   AI_RAW_7801.___________0020_1 := false;
   AI_RAW_7801.RAW_MIN := -6000;
   AI_RAW_7801.RAW_MAX := 13000;
   AI_RAW_7801.RAW_DESC := 'Thermal Resistance - 4-wire (Ni100 climate - 618)';
   AI_RAW_7801.___________0030_1 := false;
   AI_RAW_7801.___________0030_2 := false;
   AI_RAW_7801.PARAM_TYPE := 16#07;
   AI_RAW_7801.PARAM_RANGE := 16#01;
   AI_RAW_7801.PARAM_COEF := 16#08;
   AI_RAW_7801.___________0040_1 := false;
   AI_RAW_7801.___________0040_2 := false;
   AI_RAW_7801.VALUE_COEF := 0.00618;
   AI_RAW_7901.revInfo.REV_BLOCK := 'UT00801';
   AI_RAW_7901.revInfo.REV_NUMBER := '001.000';
   AI_RAW_7901.revInfo.REV_DATE := '2024-04-09';
   AI_RAW_7901.revInfo.REV_AUTHOR := 'M. Gledhill';
   AI_RAW_7901.___________0010_0 := false;
   AI_RAW_7901.___________0010_1 := false;
   AI_RAW_7901.AI_CODE := 16#7901;
   AI_RAW_7901.___________0020_0 := false;
   AI_RAW_7901.___________0020_1 := false;
   AI_RAW_7901.RAW_MIN := -6000;
   AI_RAW_7901.RAW_MAX := 13000;
   AI_RAW_7901.RAW_DESC := 'Thermal Resistance - 4-wire (Ni100 climate - 672)';
   AI_RAW_7901.___________0030_1 := false;
   AI_RAW_7901.___________0030_2 := false;
   AI_RAW_7901.PARAM_TYPE := 16#07;
   AI_RAW_7901.PARAM_RANGE := 16#01;
   AI_RAW_7901.PARAM_COEF := 16#09;
   AI_RAW_7901.___________0040_1 := false;
   AI_RAW_7901.___________0040_2 := false;
   AI_RAW_7901.VALUE_COEF := 0.00672;
   AI_RAW_7703.revInfo.REV_BLOCK := 'UT00801';
   AI_RAW_7703.revInfo.REV_NUMBER := '001.000';
   AI_RAW_7703.revInfo.REV_DATE := '2024-04-09';
   AI_RAW_7703.revInfo.REV_AUTHOR := 'M. Gledhill';
   AI_RAW_7703.___________0010_0 := false;
   AI_RAW_7703.___________0010_1 := false;
   AI_RAW_7703.AI_CODE := 16#7703;
   AI_RAW_7703.___________0020_0 := false;
   AI_RAW_7703.___________0020_1 := false;
   AI_RAW_7703.RAW_MIN := -600;
   AI_RAW_7703.RAW_MAX := 1800;
   AI_RAW_7703.RAW_DESC := 'Thermal Resistance - 4-wire (Ni100 standard - 617)';
   AI_RAW_7703.___________0030_1 := false;
   AI_RAW_7703.___________0030_2 := false;
   AI_RAW_7703.PARAM_TYPE := 16#07;
   AI_RAW_7703.PARAM_RANGE := 16#03;
   AI_RAW_7703.PARAM_COEF := 16#07;
   AI_RAW_7703.___________0040_1 := false;
   AI_RAW_7703.___________0040_2 := false;
   AI_RAW_7703.VALUE_COEF := 0.00617;
   AI_RAW_7803.revInfo.REV_BLOCK := 'UT00801';
   AI_RAW_7803.revInfo.REV_NUMBER := '001.000';
   AI_RAW_7803.revInfo.REV_DATE := '2024-04-09';
   AI_RAW_7803.revInfo.REV_AUTHOR := 'M. Gledhill';
   AI_RAW_7803.___________0010_0 := false;
   AI_RAW_7803.___________0010_1 := false;
   AI_RAW_7803.AI_CODE := 16#7803;
   AI_RAW_7803.___________0020_0 := false;
   AI_RAW_7803.___________0020_1 := false;
   AI_RAW_7803.RAW_MIN := -600;
   AI_RAW_7803.RAW_MAX := 2500;
   AI_RAW_7803.RAW_DESC := 'Thermal Resistance - 4-wire (Ni100 standard - 618)';
   AI_RAW_7803.___________0030_1 := false;
   AI_RAW_7803.___________0030_2 := false;
   AI_RAW_7803.PARAM_TYPE := 16#07;
   AI_RAW_7803.PARAM_RANGE := 16#03;
   AI_RAW_7803.PARAM_COEF := 16#08;
   AI_RAW_7803.___________0040_1 := false;
   AI_RAW_7803.___________0040_2 := false;
   AI_RAW_7803.VALUE_COEF := 0.00618;
   AI_RAW_7903.revInfo.REV_BLOCK := 'UT00801';
   AI_RAW_7903.revInfo.REV_NUMBER := '001.000';
   AI_RAW_7903.revInfo.REV_DATE := '2024-04-09';
   AI_RAW_7903.revInfo.REV_AUTHOR := 'M. Gledhill';
   AI_RAW_7903.___________0010_0 := false;
   AI_RAW_7903.___________0010_1 := false;
   AI_RAW_7903.AI_CODE := 16#7903;
   AI_RAW_7903.___________0020_0 := false;
   AI_RAW_7903.___________0020_1 := false;
   AI_RAW_7903.RAW_MIN := -600;
   AI_RAW_7903.RAW_MAX := 2500;
   AI_RAW_7903.RAW_DESC := 'Thermal Resistance - 4-wire (Ni100 standard - 672)';
   AI_RAW_7903.___________0030_1 := false;
   AI_RAW_7903.___________0030_2 := false;
   AI_RAW_7903.PARAM_TYPE := 16#07;
   AI_RAW_7903.PARAM_RANGE := 16#03;
   AI_RAW_7903.PARAM_COEF := 16#09;
   AI_RAW_7903.___________0040_1 := false;
   AI_RAW_7903.___________0040_2 := false;
   AI_RAW_7903.VALUE_COEF := 0.00672;
   AI_RAW_7711.revInfo.REV_BLOCK := 'UT00801';
   AI_RAW_7711.revInfo.REV_NUMBER := '001.000';
   AI_RAW_7711.revInfo.REV_DATE := '2024-04-09';
   AI_RAW_7711.revInfo.REV_AUTHOR := 'M. Gledhill';
   AI_RAW_7711.___________0010_0 := false;
   AI_RAW_7711.___________0010_1 := false;
   AI_RAW_7711.AI_CODE := 16#7711;
   AI_RAW_7711.___________0020_0 := false;
   AI_RAW_7711.___________0020_1 := false;
   AI_RAW_7711.RAW_MIN := -6000;
   AI_RAW_7711.RAW_MAX := 13000;
   AI_RAW_7711.RAW_DESC := 'Thermal Resistance - 4-wire (Ni200 climate - 617)';
   AI_RAW_7711.___________0030_1 := false;
   AI_RAW_7711.___________0030_2 := false;
   AI_RAW_7711.PARAM_TYPE := 16#07;
   AI_RAW_7711.PARAM_RANGE := 16#11;
   AI_RAW_7711.PARAM_COEF := 16#07;
   AI_RAW_7711.___________0040_1 := false;
   AI_RAW_7711.___________0040_2 := false;
   AI_RAW_7711.VALUE_COEF := 0.00617;
   AI_RAW_7811.revInfo.REV_BLOCK := 'UT00801';
   AI_RAW_7811.revInfo.REV_NUMBER := '001.000';
   AI_RAW_7811.revInfo.REV_DATE := '2024-04-09';
   AI_RAW_7811.revInfo.REV_AUTHOR := 'M. Gledhill';
   AI_RAW_7811.___________0010_0 := false;
   AI_RAW_7811.___________0010_1 := false;
   AI_RAW_7811.AI_CODE := 16#7811;
   AI_RAW_7811.___________0020_0 := false;
   AI_RAW_7811.___________0020_1 := false;
   AI_RAW_7811.RAW_MIN := -6000;
   AI_RAW_7811.RAW_MAX := 13000;
   AI_RAW_7811.RAW_DESC := 'Thermal Resistance - 4-wire (Ni200 climate - 618)';
   AI_RAW_7811.___________0030_1 := false;
   AI_RAW_7811.___________0030_2 := false;
   AI_RAW_7811.PARAM_TYPE := 16#07;
   AI_RAW_7811.PARAM_RANGE := 16#11;
   AI_RAW_7811.PARAM_COEF := 16#08;
   AI_RAW_7811.___________0040_1 := false;
   AI_RAW_7811.___________0040_2 := false;
   AI_RAW_7811.VALUE_COEF := 0.00618;
   AI_RAW_7911.revInfo.REV_BLOCK := 'UT00801';
   AI_RAW_7911.revInfo.REV_NUMBER := '001.000';
   AI_RAW_7911.revInfo.REV_DATE := '2024-04-09';
   AI_RAW_7911.revInfo.REV_AUTHOR := 'M. Gledhill';
   AI_RAW_7911.___________0010_0 := false;
   AI_RAW_7911.___________0010_1 := false;
   AI_RAW_7911.AI_CODE := 16#7911;
   AI_RAW_7911.___________0020_0 := false;
   AI_RAW_7911.___________0020_1 := false;
   AI_RAW_7911.RAW_MIN := -6000;
   AI_RAW_7911.RAW_MAX := 13000;
   AI_RAW_7911.RAW_DESC := 'Thermal Resistance - 4-wire (Ni200 climate - 672)';
   AI_RAW_7911.___________0030_1 := false;
   AI_RAW_7911.___________0030_2 := false;
   AI_RAW_7911.PARAM_TYPE := 16#07;
   AI_RAW_7911.PARAM_RANGE := 16#11;
   AI_RAW_7911.PARAM_COEF := 16#09;
   AI_RAW_7911.___________0040_1 := false;
   AI_RAW_7911.___________0040_2 := false;
   AI_RAW_7911.VALUE_COEF := 0.00672;
   AI_RAW_7710.revInfo.REV_BLOCK := 'UT00801';
   AI_RAW_7710.revInfo.REV_NUMBER := '001.000';
   AI_RAW_7710.revInfo.REV_DATE := '2024-04-09';
   AI_RAW_7710.revInfo.REV_AUTHOR := 'M. Gledhill';
   AI_RAW_7710.___________0010_0 := false;
   AI_RAW_7710.___________0010_1 := false;
   AI_RAW_7710.AI_CODE := 16#7710;
   AI_RAW_7710.___________0020_0 := false;
   AI_RAW_7710.___________0020_1 := false;
   AI_RAW_7710.RAW_MIN := -600;
   AI_RAW_7710.RAW_MAX := 1800;
   AI_RAW_7710.RAW_DESC := 'Thermal Resistance - 4-wire (Ni200 standard - 617)';
   AI_RAW_7710.___________0030_1 := false;
   AI_RAW_7710.___________0030_2 := false;
   AI_RAW_7710.PARAM_TYPE := 16#07;
   AI_RAW_7710.PARAM_RANGE := 16#10;
   AI_RAW_7710.PARAM_COEF := 16#07;
   AI_RAW_7710.___________0040_1 := false;
   AI_RAW_7710.___________0040_2 := false;
   AI_RAW_7710.VALUE_COEF := 0.00617;
   AI_RAW_7810.revInfo.REV_BLOCK := 'UT00801';
   AI_RAW_7810.revInfo.REV_NUMBER := '001.000';
   AI_RAW_7810.revInfo.REV_DATE := '2024-04-09';
   AI_RAW_7810.revInfo.REV_AUTHOR := 'M. Gledhill';
   AI_RAW_7810.___________0010_0 := false;
   AI_RAW_7810.___________0010_1 := false;
   AI_RAW_7810.AI_CODE := 16#7810;
   AI_RAW_7810.___________0020_0 := false;
   AI_RAW_7810.___________0020_1 := false;
   AI_RAW_7810.RAW_MIN := -600;
   AI_RAW_7810.RAW_MAX := 2500;
   AI_RAW_7810.RAW_DESC := 'Thermal Resistance - 4-wire (Ni200 standard - 618)';
   AI_RAW_7810.___________0030_1 := false;
   AI_RAW_7810.___________0030_2 := false;
   AI_RAW_7810.PARAM_TYPE := 16#07;
   AI_RAW_7810.PARAM_RANGE := 16#10;
   AI_RAW_7810.PARAM_COEF := 16#08;
   AI_RAW_7810.___________0040_1 := false;
   AI_RAW_7810.___________0040_2 := false;
   AI_RAW_7810.VALUE_COEF := 0.00618;
   AI_RAW_7910.revInfo.REV_BLOCK := 'UT00801';
   AI_RAW_7910.revInfo.REV_NUMBER := '001.000';
   AI_RAW_7910.revInfo.REV_DATE := '2024-04-09';
   AI_RAW_7910.revInfo.REV_AUTHOR := 'M. Gledhill';
   AI_RAW_7910.___________0010_0 := false;
   AI_RAW_7910.___________0010_1 := false;
   AI_RAW_7910.AI_CODE := 16#7910;
   AI_RAW_7910.___________0020_0 := false;
   AI_RAW_7910.___________0020_1 := false;
   AI_RAW_7910.RAW_MIN := -600;
   AI_RAW_7910.RAW_MAX := 2500;
   AI_RAW_7910.RAW_DESC := 'Thermal Resistance - 4-wire (Ni200 standard - 672)';
   AI_RAW_7910.___________0030_1 := false;
   AI_RAW_7910.___________0030_2 := false;
   AI_RAW_7910.PARAM_TYPE := 16#07;
   AI_RAW_7910.PARAM_RANGE := 16#10;
   AI_RAW_7910.PARAM_COEF := 16#09;
   AI_RAW_7910.___________0040_1 := false;
   AI_RAW_7910.___________0040_2 := false;
   AI_RAW_7910.VALUE_COEF := 0.00672;
   AI_RAW_7713.revInfo.REV_BLOCK := 'UT00801';
   AI_RAW_7713.revInfo.REV_NUMBER := '001.000';
   AI_RAW_7713.revInfo.REV_DATE := '2024-04-09';
   AI_RAW_7713.revInfo.REV_AUTHOR := 'M. Gledhill';
   AI_RAW_7713.___________0010_0 := false;
   AI_RAW_7713.___________0010_1 := false;
   AI_RAW_7713.AI_CODE := 16#7713;
   AI_RAW_7713.___________0020_0 := false;
   AI_RAW_7713.___________0020_1 := false;
   AI_RAW_7713.RAW_MIN := -6000;
   AI_RAW_7713.RAW_MAX := 13000;
   AI_RAW_7713.RAW_DESC := 'Thermal Resistance - 4-wire (Ni500 climate - 617)';
   AI_RAW_7713.___________0030_1 := false;
   AI_RAW_7713.___________0030_2 := false;
   AI_RAW_7713.PARAM_TYPE := 16#07;
   AI_RAW_7713.PARAM_RANGE := 16#13;
   AI_RAW_7713.PARAM_COEF := 16#07;
   AI_RAW_7713.___________0040_1 := false;
   AI_RAW_7713.___________0040_2 := false;
   AI_RAW_7713.VALUE_COEF := 0.00617;
   AI_RAW_7813.revInfo.REV_BLOCK := 'UT00801';
   AI_RAW_7813.revInfo.REV_NUMBER := '001.000';
   AI_RAW_7813.revInfo.REV_DATE := '2024-04-09';
   AI_RAW_7813.revInfo.REV_AUTHOR := 'M. Gledhill';
   AI_RAW_7813.___________0010_0 := false;
   AI_RAW_7813.___________0010_1 := false;
   AI_RAW_7813.AI_CODE := 16#7813;
   AI_RAW_7813.___________0020_0 := false;
   AI_RAW_7813.___________0020_1 := false;
   AI_RAW_7813.RAW_MIN := -6000;
   AI_RAW_7813.RAW_MAX := 13000;
   AI_RAW_7813.RAW_DESC := 'Thermal Resistance - 4-wire (Ni500 climate - 618)';
   AI_RAW_7813.___________0030_1 := false;
   AI_RAW_7813.___________0030_2 := false;
   AI_RAW_7813.PARAM_TYPE := 16#07;
   AI_RAW_7813.PARAM_RANGE := 16#13;
   AI_RAW_7813.PARAM_COEF := 16#08;
   AI_RAW_7813.___________0040_1 := false;
   AI_RAW_7813.___________0040_2 := false;
   AI_RAW_7813.VALUE_COEF := 0.00618;
   AI_RAW_7913.revInfo.REV_BLOCK := 'UT00801';
   AI_RAW_7913.revInfo.REV_NUMBER := '001.000';
   AI_RAW_7913.revInfo.REV_DATE := '2024-04-09';
   AI_RAW_7913.revInfo.REV_AUTHOR := 'M. Gledhill';
   AI_RAW_7913.___________0010_0 := false;
   AI_RAW_7913.___________0010_1 := false;
   AI_RAW_7913.AI_CODE := 16#7913;
   AI_RAW_7913.___________0020_0 := false;
   AI_RAW_7913.___________0020_1 := false;
   AI_RAW_7913.RAW_MIN := -6000;
   AI_RAW_7913.RAW_MAX := 13000;
   AI_RAW_7913.RAW_DESC := 'Thermal Resistance - 4-wire (Ni500 climate - 672)';
   AI_RAW_7913.___________0030_1 := false;
   AI_RAW_7913.___________0030_2 := false;
   AI_RAW_7913.PARAM_TYPE := 16#07;
   AI_RAW_7913.PARAM_RANGE := 16#13;
   AI_RAW_7913.PARAM_COEF := 16#09;
   AI_RAW_7913.___________0040_1 := false;
   AI_RAW_7913.___________0040_2 := false;
   AI_RAW_7913.VALUE_COEF := 0.00672;
   AI_RAW_7712.revInfo.REV_BLOCK := 'UT00801';
   AI_RAW_7712.revInfo.REV_NUMBER := '001.000';
   AI_RAW_7712.revInfo.REV_DATE := '2024-04-09';
   AI_RAW_7712.revInfo.REV_AUTHOR := 'M. Gledhill';
   AI_RAW_7712.___________0010_0 := false;
   AI_RAW_7712.___________0010_1 := false;
   AI_RAW_7712.AI_CODE := 16#7712;
   AI_RAW_7712.___________0020_0 := false;
   AI_RAW_7712.___________0020_1 := false;
   AI_RAW_7712.RAW_MIN := -600;
   AI_RAW_7712.RAW_MAX := 1800;
   AI_RAW_7712.RAW_DESC := 'Thermal Resistance - 4-wire (Ni500 standard - 617)';
   AI_RAW_7712.___________0030_1 := false;
   AI_RAW_7712.___________0030_2 := false;
   AI_RAW_7712.PARAM_TYPE := 16#07;
   AI_RAW_7712.PARAM_RANGE := 16#12;
   AI_RAW_7712.PARAM_COEF := 16#07;
   AI_RAW_7712.___________0040_1 := false;
   AI_RAW_7712.___________0040_2 := false;
   AI_RAW_7712.VALUE_COEF := 0.00617;
   AI_RAW_7812.revInfo.REV_BLOCK := 'UT00801';
   AI_RAW_7812.revInfo.REV_NUMBER := '001.000';
   AI_RAW_7812.revInfo.REV_DATE := '2024-04-09';
   AI_RAW_7812.revInfo.REV_AUTHOR := 'M. Gledhill';
   AI_RAW_7812.___________0010_0 := false;
   AI_RAW_7812.___________0010_1 := false;
   AI_RAW_7812.AI_CODE := 16#7812;
   AI_RAW_7812.___________0020_0 := false;
   AI_RAW_7812.___________0020_1 := false;
   AI_RAW_7812.RAW_MIN := -600;
   AI_RAW_7812.RAW_MAX := 2500;
   AI_RAW_7812.RAW_DESC := 'Thermal Resistance - 4-wire (Ni500 standard - 618)';
   AI_RAW_7812.___________0030_1 := false;
   AI_RAW_7812.___________0030_2 := false;
   AI_RAW_7812.PARAM_TYPE := 16#07;
   AI_RAW_7812.PARAM_RANGE := 16#12;
   AI_RAW_7812.PARAM_COEF := 16#08;
   AI_RAW_7812.___________0040_1 := false;
   AI_RAW_7812.___________0040_2 := false;
   AI_RAW_7812.VALUE_COEF := 0.00618;
   AI_RAW_7912.revInfo.REV_BLOCK := 'UT00801';
   AI_RAW_7912.revInfo.REV_NUMBER := '001.000';
   AI_RAW_7912.revInfo.REV_DATE := '2024-04-09';
   AI_RAW_7912.revInfo.REV_AUTHOR := 'M. Gledhill';
   AI_RAW_7912.___________0010_0 := false;
   AI_RAW_7912.___________0010_1 := false;
   AI_RAW_7912.AI_CODE := 16#7912;
   AI_RAW_7912.___________0020_0 := false;
   AI_RAW_7912.___________0020_1 := false;
   AI_RAW_7912.RAW_MIN := -600;
   AI_RAW_7912.RAW_MAX := 2500;
   AI_RAW_7912.RAW_DESC := 'Thermal Resistance - 4-wire (Ni500 standard - 672)';
   AI_RAW_7912.___________0030_1 := false;
   AI_RAW_7912.___________0030_2 := false;
   AI_RAW_7912.PARAM_TYPE := 16#07;
   AI_RAW_7912.PARAM_RANGE := 16#12;
   AI_RAW_7912.PARAM_COEF := 16#09;
   AI_RAW_7912.___________0040_1 := false;
   AI_RAW_7912.___________0040_2 := false;
   AI_RAW_7912.VALUE_COEF := 0.00672;
   AI_RAW_770A.revInfo.REV_BLOCK := 'UT00801';
   AI_RAW_770A.revInfo.REV_NUMBER := '001.000';
   AI_RAW_770A.revInfo.REV_DATE := '2024-04-09';
   AI_RAW_770A.revInfo.REV_AUTHOR := 'M. Gledhill';
   AI_RAW_770A.___________0010_0 := false;
   AI_RAW_770A.___________0010_1 := false;
   AI_RAW_770A.AI_CODE := 16#770A;
   AI_RAW_770A.___________0020_0 := false;
   AI_RAW_770A.___________0020_1 := false;
   AI_RAW_770A.RAW_MIN := -6000;
   AI_RAW_770A.RAW_MAX := 13000;
   AI_RAW_770A.RAW_DESC := 'Thermal Resistance - 4-wire (Ni1000 climate - 617)';
   AI_RAW_770A.___________0030_1 := false;
   AI_RAW_770A.___________0030_2 := false;
   AI_RAW_770A.PARAM_TYPE := 16#07;
   AI_RAW_770A.PARAM_RANGE := 16#0A;
   AI_RAW_770A.PARAM_COEF := 16#07;
   AI_RAW_770A.___________0040_1 := false;
   AI_RAW_770A.___________0040_2 := false;
   AI_RAW_770A.VALUE_COEF := 0.00617;
   AI_RAW_780A.revInfo.REV_BLOCK := 'UT00801';
   AI_RAW_780A.revInfo.REV_NUMBER := '001.000';
   AI_RAW_780A.revInfo.REV_DATE := '2024-04-09';
   AI_RAW_780A.revInfo.REV_AUTHOR := 'M. Gledhill';
   AI_RAW_780A.___________0010_0 := false;
   AI_RAW_780A.___________0010_1 := false;
   AI_RAW_780A.AI_CODE := 16#780A;
   AI_RAW_780A.___________0020_0 := false;
   AI_RAW_780A.___________0020_1 := false;
   AI_RAW_780A.RAW_MIN := -6000;
   AI_RAW_780A.RAW_MAX := 13000;
   AI_RAW_780A.RAW_DESC := 'Thermal Resistance - 4-wire (Ni1000 climate - 618)';
   AI_RAW_780A.___________0030_1 := false;
   AI_RAW_780A.___________0030_2 := false;
   AI_RAW_780A.PARAM_TYPE := 16#07;
   AI_RAW_780A.PARAM_RANGE := 16#0A;
   AI_RAW_780A.PARAM_COEF := 16#08;
   AI_RAW_780A.___________0040_1 := false;
   AI_RAW_780A.___________0040_2 := false;
   AI_RAW_780A.VALUE_COEF := 0.00618;
   AI_RAW_790A.revInfo.REV_BLOCK := 'UT00801';
   AI_RAW_790A.revInfo.REV_NUMBER := '001.000';
   AI_RAW_790A.revInfo.REV_DATE := '2024-04-09';
   AI_RAW_790A.revInfo.REV_AUTHOR := 'M. Gledhill';
   AI_RAW_790A.___________0010_0 := false;
   AI_RAW_790A.___________0010_1 := false;
   AI_RAW_790A.AI_CODE := 16#790A;
   AI_RAW_790A.___________0020_0 := false;
   AI_RAW_790A.___________0020_1 := false;
   AI_RAW_790A.RAW_MIN := -6000;
   AI_RAW_790A.RAW_MAX := 13000;
   AI_RAW_790A.RAW_DESC := 'Thermal Resistance - 4-wire (Ni1000 climate - 672)';
   AI_RAW_790A.___________0030_1 := false;
   AI_RAW_790A.___________0030_2 := false;
   AI_RAW_790A.PARAM_TYPE := 16#07;
   AI_RAW_790A.PARAM_RANGE := 16#0A;
   AI_RAW_790A.PARAM_COEF := 16#09;
   AI_RAW_790A.___________0040_1 := false;
   AI_RAW_790A.___________0040_2 := false;
   AI_RAW_790A.VALUE_COEF := 0.00672;
   AI_RAW_7706.revInfo.REV_BLOCK := 'UT00801';
   AI_RAW_7706.revInfo.REV_NUMBER := '001.000';
   AI_RAW_7706.revInfo.REV_DATE := '2024-04-09';
   AI_RAW_7706.revInfo.REV_AUTHOR := 'M. Gledhill';
   AI_RAW_7706.___________0010_0 := false;
   AI_RAW_7706.___________0010_1 := false;
   AI_RAW_7706.AI_CODE := 16#7706;
   AI_RAW_7706.___________0020_0 := false;
   AI_RAW_7706.___________0020_1 := false;
   AI_RAW_7706.RAW_MIN := -600;
   AI_RAW_7706.RAW_MAX := 1800;
   AI_RAW_7706.RAW_DESC := 'Thermal Resistance - 4-wire (Ni1000 standard - 617)';
   AI_RAW_7706.___________0030_1 := false;
   AI_RAW_7706.___________0030_2 := false;
   AI_RAW_7706.PARAM_TYPE := 16#07;
   AI_RAW_7706.PARAM_RANGE := 16#06;
   AI_RAW_7706.PARAM_COEF := 16#07;
   AI_RAW_7706.___________0040_1 := false;
   AI_RAW_7706.___________0040_2 := false;
   AI_RAW_7706.VALUE_COEF := 0.00617;
   AI_RAW_7806.revInfo.REV_BLOCK := 'UT00801';
   AI_RAW_7806.revInfo.REV_NUMBER := '001.000';
   AI_RAW_7806.revInfo.REV_DATE := '2024-04-09';
   AI_RAW_7806.revInfo.REV_AUTHOR := 'M. Gledhill';
   AI_RAW_7806.___________0010_0 := false;
   AI_RAW_7806.___________0010_1 := false;
   AI_RAW_7806.AI_CODE := 16#7806;
   AI_RAW_7806.___________0020_0 := false;
   AI_RAW_7806.___________0020_1 := false;
   AI_RAW_7806.RAW_MIN := -600;
   AI_RAW_7806.RAW_MAX := 2500;
   AI_RAW_7806.RAW_DESC := 'Thermal Resistance - 4-wire (Ni1000 standard - 618)';
   AI_RAW_7806.___________0030_1 := false;
   AI_RAW_7806.___________0030_2 := false;
   AI_RAW_7806.PARAM_TYPE := 16#07;
   AI_RAW_7806.PARAM_RANGE := 16#06;
   AI_RAW_7806.PARAM_COEF := 16#08;
   AI_RAW_7806.___________0040_1 := false;
   AI_RAW_7806.___________0040_2 := false;
   AI_RAW_7806.VALUE_COEF := 0.00618;
   AI_RAW_7906.revInfo.REV_BLOCK := 'UT00801';
   AI_RAW_7906.revInfo.REV_NUMBER := '001.000';
   AI_RAW_7906.revInfo.REV_DATE := '2024-04-09';
   AI_RAW_7906.revInfo.REV_AUTHOR := 'M. Gledhill';
   AI_RAW_7906.___________0010_0 := false;
   AI_RAW_7906.___________0010_1 := false;
   AI_RAW_7906.AI_CODE := 16#7906;
   AI_RAW_7906.___________0020_0 := false;
   AI_RAW_7906.___________0020_1 := false;
   AI_RAW_7906.RAW_MIN := -600;
   AI_RAW_7906.RAW_MAX := 2500;
   AI_RAW_7906.RAW_DESC := 'Thermal Resistance - 4-wire (Ni1000 standard - 672)';
   AI_RAW_7906.___________0030_1 := false;
   AI_RAW_7906.___________0030_2 := false;
   AI_RAW_7906.PARAM_TYPE := 16#07;
   AI_RAW_7906.PARAM_RANGE := 16#06;
   AI_RAW_7906.PARAM_COEF := 16#09;
   AI_RAW_7906.___________0040_1 := false;
   AI_RAW_7906.___________0040_2 := false;
   AI_RAW_7906.VALUE_COEF := 0.00672;
   AI_RAW_7015.revInfo.REV_BLOCK := 'UT00801';
   AI_RAW_7015.revInfo.REV_NUMBER := '001.000';
   AI_RAW_7015.revInfo.REV_DATE := '2024-04-09';
   AI_RAW_7015.revInfo.REV_AUTHOR := 'M. Gledhill';
   AI_RAW_7015.___________0010_0 := false;
   AI_RAW_7015.___________0010_1 := false;
   AI_RAW_7015.AI_CODE := 16#7015;
   AI_RAW_7015.___________0020_0 := false;
   AI_RAW_7015.___________0020_1 := false;
   AI_RAW_7015.RAW_MIN := -12000;
   AI_RAW_7015.RAW_MAX := 13000;
   AI_RAW_7015.RAW_DESC := 'Thermal Resistance - 4-wire (Pt10 climate - 3851)';
   AI_RAW_7015.___________0030_1 := false;
   AI_RAW_7015.___________0030_2 := false;
   AI_RAW_7015.PARAM_TYPE := 16#07;
   AI_RAW_7015.PARAM_RANGE := 16#15;
   AI_RAW_7015.PARAM_COEF := 16#00;
   AI_RAW_7015.___________0040_1 := false;
   AI_RAW_7015.___________0040_2 := false;
   AI_RAW_7015.VALUE_COEF := 0.003851;
   AI_RAW_7215.revInfo.REV_BLOCK := 'UT00801';
   AI_RAW_7215.revInfo.REV_NUMBER := '001.000';
   AI_RAW_7215.revInfo.REV_DATE := '2024-04-09';
   AI_RAW_7215.revInfo.REV_AUTHOR := 'M. Gledhill';
   AI_RAW_7215.___________0010_0 := false;
   AI_RAW_7215.___________0010_1 := false;
   AI_RAW_7215.AI_CODE := 16#7215;
   AI_RAW_7215.___________0020_0 := false;
   AI_RAW_7215.___________0020_1 := false;
   AI_RAW_7215.RAW_MIN := -12000;
   AI_RAW_7215.RAW_MAX := 13000;
   AI_RAW_7215.RAW_DESC := 'Thermal Resistance - 4-wire (Pt10 climate - 3902)';
   AI_RAW_7215.___________0030_1 := false;
   AI_RAW_7215.___________0030_2 := false;
   AI_RAW_7215.PARAM_TYPE := 16#07;
   AI_RAW_7215.PARAM_RANGE := 16#15;
   AI_RAW_7215.PARAM_COEF := 16#02;
   AI_RAW_7215.___________0040_1 := false;
   AI_RAW_7215.___________0040_2 := false;
   AI_RAW_7215.VALUE_COEF := 0.003902;
   AI_RAW_7515.revInfo.REV_BLOCK := 'UT00801';
   AI_RAW_7515.revInfo.REV_NUMBER := '001.000';
   AI_RAW_7515.revInfo.REV_DATE := '2024-04-09';
   AI_RAW_7515.revInfo.REV_AUTHOR := 'M. Gledhill';
   AI_RAW_7515.___________0010_0 := false;
   AI_RAW_7515.___________0010_1 := false;
   AI_RAW_7515.AI_CODE := 16#7515;
   AI_RAW_7515.___________0020_0 := false;
   AI_RAW_7515.___________0020_1 := false;
   AI_RAW_7515.RAW_MIN := -12000;
   AI_RAW_7515.RAW_MAX := 13000;
   AI_RAW_7515.RAW_DESC := 'Thermal Resistance - 4-wire (Pt10 climate - 391)';
   AI_RAW_7515.___________0030_1 := false;
   AI_RAW_7515.___________0030_2 := false;
   AI_RAW_7515.PARAM_TYPE := 16#07;
   AI_RAW_7515.PARAM_RANGE := 16#15;
   AI_RAW_7515.PARAM_COEF := 16#05;
   AI_RAW_7515.___________0040_1 := false;
   AI_RAW_7515.___________0040_2 := false;
   AI_RAW_7515.VALUE_COEF := 0.00391;
   AI_RAW_7115.revInfo.REV_BLOCK := 'UT00801';
   AI_RAW_7115.revInfo.REV_NUMBER := '001.000';
   AI_RAW_7115.revInfo.REV_DATE := '2024-04-09';
   AI_RAW_7115.revInfo.REV_AUTHOR := 'M. Gledhill';
   AI_RAW_7115.___________0010_0 := false;
   AI_RAW_7115.___________0010_1 := false;
   AI_RAW_7115.AI_CODE := 16#7115;
   AI_RAW_7115.___________0020_0 := false;
   AI_RAW_7115.___________0020_1 := false;
   AI_RAW_7115.RAW_MIN := -12000;
   AI_RAW_7115.RAW_MAX := 13000;
   AI_RAW_7115.RAW_DESC := 'Thermal Resistance - 4-wire (Pt10 climate - 3916)';
   AI_RAW_7115.___________0030_1 := false;
   AI_RAW_7115.___________0030_2 := false;
   AI_RAW_7115.PARAM_TYPE := 16#07;
   AI_RAW_7115.PARAM_RANGE := 16#15;
   AI_RAW_7115.PARAM_COEF := 16#01;
   AI_RAW_7115.___________0040_1 := false;
   AI_RAW_7115.___________0040_2 := false;
   AI_RAW_7115.VALUE_COEF := 0.003916;
   AI_RAW_7315.revInfo.REV_BLOCK := 'UT00801';
   AI_RAW_7315.revInfo.REV_NUMBER := '001.000';
   AI_RAW_7315.revInfo.REV_DATE := '2024-04-09';
   AI_RAW_7315.revInfo.REV_AUTHOR := 'M. Gledhill';
   AI_RAW_7315.___________0010_0 := false;
   AI_RAW_7315.___________0010_1 := false;
   AI_RAW_7315.AI_CODE := 16#7315;
   AI_RAW_7315.___________0020_0 := false;
   AI_RAW_7315.___________0020_1 := false;
   AI_RAW_7315.RAW_MIN := -12000;
   AI_RAW_7315.RAW_MAX := 13000;
   AI_RAW_7315.RAW_DESC := 'Thermal Resistance - 4-wire (Pt10 climate - 392)';
   AI_RAW_7315.___________0030_1 := false;
   AI_RAW_7315.___________0030_2 := false;
   AI_RAW_7315.PARAM_TYPE := 16#07;
   AI_RAW_7315.PARAM_RANGE := 16#15;
   AI_RAW_7315.PARAM_COEF := 16#03;
   AI_RAW_7315.___________0040_1 := false;
   AI_RAW_7315.___________0040_2 := false;
   AI_RAW_7315.VALUE_COEF := 0.00392;
   AI_RAW_7014.revInfo.REV_BLOCK := 'UT00801';
   AI_RAW_7014.revInfo.REV_NUMBER := '001.000';
   AI_RAW_7014.revInfo.REV_DATE := '2024-04-09';
   AI_RAW_7014.revInfo.REV_AUTHOR := 'M. Gledhill';
   AI_RAW_7014.___________0010_0 := false;
   AI_RAW_7014.___________0010_1 := false;
   AI_RAW_7014.AI_CODE := 16#7014;
   AI_RAW_7014.___________0020_0 := false;
   AI_RAW_7014.___________0020_1 := false;
   AI_RAW_7014.RAW_MIN := -2000;
   AI_RAW_7014.RAW_MAX := 8500;
   AI_RAW_7014.RAW_DESC := 'Thermal Resistance - 4-wire (Pt10 standard - 3851)';
   AI_RAW_7014.___________0030_1 := false;
   AI_RAW_7014.___________0030_2 := false;
   AI_RAW_7014.PARAM_TYPE := 16#07;
   AI_RAW_7014.PARAM_RANGE := 16#14;
   AI_RAW_7014.PARAM_COEF := 16#00;
   AI_RAW_7014.___________0040_1 := false;
   AI_RAW_7014.___________0040_2 := false;
   AI_RAW_7014.VALUE_COEF := 0.003851;
   AI_RAW_7214.revInfo.REV_BLOCK := 'UT00801';
   AI_RAW_7214.revInfo.REV_NUMBER := '001.000';
   AI_RAW_7214.revInfo.REV_DATE := '2024-04-09';
   AI_RAW_7214.revInfo.REV_AUTHOR := 'M. Gledhill';
   AI_RAW_7214.___________0010_0 := false;
   AI_RAW_7214.___________0010_1 := false;
   AI_RAW_7214.AI_CODE := 16#7214;
   AI_RAW_7214.___________0020_0 := false;
   AI_RAW_7214.___________0020_1 := false;
   AI_RAW_7214.RAW_MIN := -2000;
   AI_RAW_7214.RAW_MAX := 8500;
   AI_RAW_7214.RAW_DESC := 'Thermal Resistance - 4-wire (Pt10 standard - 3902)';
   AI_RAW_7214.___________0030_1 := false;
   AI_RAW_7214.___________0030_2 := false;
   AI_RAW_7214.PARAM_TYPE := 16#07;
   AI_RAW_7214.PARAM_RANGE := 16#14;
   AI_RAW_7214.PARAM_COEF := 16#02;
   AI_RAW_7214.___________0040_1 := false;
   AI_RAW_7214.___________0040_2 := false;
   AI_RAW_7214.VALUE_COEF := 0.003902;
   AI_RAW_7514.revInfo.REV_BLOCK := 'UT00801';
   AI_RAW_7514.revInfo.REV_NUMBER := '001.000';
   AI_RAW_7514.revInfo.REV_DATE := '2024-04-09';
   AI_RAW_7514.revInfo.REV_AUTHOR := 'M. Gledhill';
   AI_RAW_7514.___________0010_0 := false;
   AI_RAW_7514.___________0010_1 := false;
   AI_RAW_7514.AI_CODE := 16#7514;
   AI_RAW_7514.___________0020_0 := false;
   AI_RAW_7514.___________0020_1 := false;
   AI_RAW_7514.RAW_MIN := -2000;
   AI_RAW_7514.RAW_MAX := 8500;
   AI_RAW_7514.RAW_DESC := 'Thermal Resistance - 4-wire (Pt10 standard - 391)';
   AI_RAW_7514.___________0030_1 := false;
   AI_RAW_7514.___________0030_2 := false;
   AI_RAW_7514.PARAM_TYPE := 16#07;
   AI_RAW_7514.PARAM_RANGE := 16#14;
   AI_RAW_7514.PARAM_COEF := 16#05;
   AI_RAW_7514.___________0040_1 := false;
   AI_RAW_7514.___________0040_2 := false;
   AI_RAW_7514.VALUE_COEF := 0.00391;
   AI_RAW_7114.revInfo.REV_BLOCK := 'UT00801';
   AI_RAW_7114.revInfo.REV_NUMBER := '001.000';
   AI_RAW_7114.revInfo.REV_DATE := '2024-04-09';
   AI_RAW_7114.revInfo.REV_AUTHOR := 'M. Gledhill';
   AI_RAW_7114.___________0010_0 := false;
   AI_RAW_7114.___________0010_1 := false;
   AI_RAW_7114.AI_CODE := 16#7114;
   AI_RAW_7114.___________0020_0 := false;
   AI_RAW_7114.___________0020_1 := false;
   AI_RAW_7114.RAW_MIN := -2000;
   AI_RAW_7114.RAW_MAX := 8500;
   AI_RAW_7114.RAW_DESC := 'Thermal Resistance - 4-wire (Pt10 standard - 3916)';
   AI_RAW_7114.___________0030_1 := false;
   AI_RAW_7114.___________0030_2 := false;
   AI_RAW_7114.PARAM_TYPE := 16#07;
   AI_RAW_7114.PARAM_RANGE := 16#14;
   AI_RAW_7114.PARAM_COEF := 16#01;
   AI_RAW_7114.___________0040_1 := false;
   AI_RAW_7114.___________0040_2 := false;
   AI_RAW_7114.VALUE_COEF := 0.003916;
   AI_RAW_7314.revInfo.REV_BLOCK := 'UT00801';
   AI_RAW_7314.revInfo.REV_NUMBER := '001.000';
   AI_RAW_7314.revInfo.REV_DATE := '2024-04-09';
   AI_RAW_7314.revInfo.REV_AUTHOR := 'M. Gledhill';
   AI_RAW_7314.___________0010_0 := false;
   AI_RAW_7314.___________0010_1 := false;
   AI_RAW_7314.AI_CODE := 16#7314;
   AI_RAW_7314.___________0020_0 := false;
   AI_RAW_7314.___________0020_1 := false;
   AI_RAW_7314.RAW_MIN := -2000;
   AI_RAW_7314.RAW_MAX := 8500;
   AI_RAW_7314.RAW_DESC := 'Thermal Resistance - 4-wire (Pt10 standard - 392)';
   AI_RAW_7314.___________0030_1 := false;
   AI_RAW_7314.___________0030_2 := false;
   AI_RAW_7314.PARAM_TYPE := 16#07;
   AI_RAW_7314.PARAM_RANGE := 16#14;
   AI_RAW_7314.PARAM_COEF := 16#03;
   AI_RAW_7314.___________0040_1 := false;
   AI_RAW_7314.___________0040_2 := false;
   AI_RAW_7314.VALUE_COEF := 0.00392;
   AI_RAW_7017.revInfo.REV_BLOCK := 'UT00801';
   AI_RAW_7017.revInfo.REV_NUMBER := '001.000';
   AI_RAW_7017.revInfo.REV_DATE := '2024-04-09';
   AI_RAW_7017.revInfo.REV_AUTHOR := 'M. Gledhill';
   AI_RAW_7017.___________0010_0 := false;
   AI_RAW_7017.___________0010_1 := false;
   AI_RAW_7017.AI_CODE := 16#7017;
   AI_RAW_7017.___________0020_0 := false;
   AI_RAW_7017.___________0020_1 := false;
   AI_RAW_7017.RAW_MIN := -12000;
   AI_RAW_7017.RAW_MAX := 13000;
   AI_RAW_7017.RAW_DESC := 'Thermal Resistance - 4-wire (Pt50 climate - 3851)';
   AI_RAW_7017.___________0030_1 := false;
   AI_RAW_7017.___________0030_2 := false;
   AI_RAW_7017.PARAM_TYPE := 16#07;
   AI_RAW_7017.PARAM_RANGE := 16#17;
   AI_RAW_7017.PARAM_COEF := 16#00;
   AI_RAW_7017.___________0040_1 := false;
   AI_RAW_7017.___________0040_2 := false;
   AI_RAW_7017.VALUE_COEF := 0.003851;
   AI_RAW_7217.revInfo.REV_BLOCK := 'UT00801';
   AI_RAW_7217.revInfo.REV_NUMBER := '001.000';
   AI_RAW_7217.revInfo.REV_DATE := '2024-04-09';
   AI_RAW_7217.revInfo.REV_AUTHOR := 'M. Gledhill';
   AI_RAW_7217.___________0010_0 := false;
   AI_RAW_7217.___________0010_1 := false;
   AI_RAW_7217.AI_CODE := 16#7217;
   AI_RAW_7217.___________0020_0 := false;
   AI_RAW_7217.___________0020_1 := false;
   AI_RAW_7217.RAW_MIN := -12000;
   AI_RAW_7217.RAW_MAX := 13000;
   AI_RAW_7217.RAW_DESC := 'Thermal Resistance - 4-wire (Pt50 climate - 3902)';
   AI_RAW_7217.___________0030_1 := false;
   AI_RAW_7217.___________0030_2 := false;
   AI_RAW_7217.PARAM_TYPE := 16#07;
   AI_RAW_7217.PARAM_RANGE := 16#17;
   AI_RAW_7217.PARAM_COEF := 16#02;
   AI_RAW_7217.___________0040_1 := false;
   AI_RAW_7217.___________0040_2 := false;
   AI_RAW_7217.VALUE_COEF := 0.003902;
   AI_RAW_7517.revInfo.REV_BLOCK := 'UT00801';
   AI_RAW_7517.revInfo.REV_NUMBER := '001.000';
   AI_RAW_7517.revInfo.REV_DATE := '2024-04-09';
   AI_RAW_7517.revInfo.REV_AUTHOR := 'M. Gledhill';
   AI_RAW_7517.___________0010_0 := false;
   AI_RAW_7517.___________0010_1 := false;
   AI_RAW_7517.AI_CODE := 16#7517;
   AI_RAW_7517.___________0020_0 := false;
   AI_RAW_7517.___________0020_1 := false;
   AI_RAW_7517.RAW_MIN := -12000;
   AI_RAW_7517.RAW_MAX := 13000;
   AI_RAW_7517.RAW_DESC := 'Thermal Resistance - 4-wire (Pt50 climate - 391)';
   AI_RAW_7517.___________0030_1 := false;
   AI_RAW_7517.___________0030_2 := false;
   AI_RAW_7517.PARAM_TYPE := 16#07;
   AI_RAW_7517.PARAM_RANGE := 16#17;
   AI_RAW_7517.PARAM_COEF := 16#05;
   AI_RAW_7517.___________0040_1 := false;
   AI_RAW_7517.___________0040_2 := false;
   AI_RAW_7517.VALUE_COEF := 0.00391;
   AI_RAW_7117.revInfo.REV_BLOCK := 'UT00801';
   AI_RAW_7117.revInfo.REV_NUMBER := '001.000';
   AI_RAW_7117.revInfo.REV_DATE := '2024-04-09';
   AI_RAW_7117.revInfo.REV_AUTHOR := 'M. Gledhill';
   AI_RAW_7117.___________0010_0 := false;
   AI_RAW_7117.___________0010_1 := false;
   AI_RAW_7117.AI_CODE := 16#7117;
   AI_RAW_7117.___________0020_0 := false;
   AI_RAW_7117.___________0020_1 := false;
   AI_RAW_7117.RAW_MIN := -12000;
   AI_RAW_7117.RAW_MAX := 13000;
   AI_RAW_7117.RAW_DESC := 'Thermal Resistance - 4-wire (Pt50 climate - 3916)';
   AI_RAW_7117.___________0030_1 := false;
   AI_RAW_7117.___________0030_2 := false;
   AI_RAW_7117.PARAM_TYPE := 16#07;
   AI_RAW_7117.PARAM_RANGE := 16#17;
   AI_RAW_7117.PARAM_COEF := 16#01;
   AI_RAW_7117.___________0040_1 := false;
   AI_RAW_7117.___________0040_2 := false;
   AI_RAW_7117.VALUE_COEF := 0.003916;
   AI_RAW_7317.revInfo.REV_BLOCK := 'UT00801';
   AI_RAW_7317.revInfo.REV_NUMBER := '001.000';
   AI_RAW_7317.revInfo.REV_DATE := '2024-04-09';
   AI_RAW_7317.revInfo.REV_AUTHOR := 'M. Gledhill';
   AI_RAW_7317.___________0010_0 := false;
   AI_RAW_7317.___________0010_1 := false;
   AI_RAW_7317.AI_CODE := 16#7317;
   AI_RAW_7317.___________0020_0 := false;
   AI_RAW_7317.___________0020_1 := false;
   AI_RAW_7317.RAW_MIN := -12000;
   AI_RAW_7317.RAW_MAX := 13000;
   AI_RAW_7317.RAW_DESC := 'Thermal Resistance - 4-wire (Pt50 climate - 392)';
   AI_RAW_7317.___________0030_1 := false;
   AI_RAW_7317.___________0030_2 := false;
   AI_RAW_7317.PARAM_TYPE := 16#07;
   AI_RAW_7317.PARAM_RANGE := 16#17;
   AI_RAW_7317.PARAM_COEF := 16#03;
   AI_RAW_7317.___________0040_1 := false;
   AI_RAW_7317.___________0040_2 := false;
   AI_RAW_7317.VALUE_COEF := 0.00392;
   AI_RAW_7016.revInfo.REV_BLOCK := 'UT00801';
   AI_RAW_7016.revInfo.REV_NUMBER := '001.000';
   AI_RAW_7016.revInfo.REV_DATE := '2024-04-09';
   AI_RAW_7016.revInfo.REV_AUTHOR := 'M. Gledhill';
   AI_RAW_7016.___________0010_0 := false;
   AI_RAW_7016.___________0010_1 := false;
   AI_RAW_7016.AI_CODE := 16#7016;
   AI_RAW_7016.___________0020_0 := false;
   AI_RAW_7016.___________0020_1 := false;
   AI_RAW_7016.RAW_MIN := -2000;
   AI_RAW_7016.RAW_MAX := 8500;
   AI_RAW_7016.RAW_DESC := 'Thermal Resistance - 4-wire (Pt50 standard - 3851)';
   AI_RAW_7016.___________0030_1 := false;
   AI_RAW_7016.___________0030_2 := false;
   AI_RAW_7016.PARAM_TYPE := 16#07;
   AI_RAW_7016.PARAM_RANGE := 16#16;
   AI_RAW_7016.PARAM_COEF := 16#00;
   AI_RAW_7016.___________0040_1 := false;
   AI_RAW_7016.___________0040_2 := false;
   AI_RAW_7016.VALUE_COEF := 0.003851;
   AI_RAW_7216.revInfo.REV_BLOCK := 'UT00801';
   AI_RAW_7216.revInfo.REV_NUMBER := '001.000';
   AI_RAW_7216.revInfo.REV_DATE := '2024-04-09';
   AI_RAW_7216.revInfo.REV_AUTHOR := 'M. Gledhill';
   AI_RAW_7216.___________0010_0 := false;
   AI_RAW_7216.___________0010_1 := false;
   AI_RAW_7216.AI_CODE := 16#7216;
   AI_RAW_7216.___________0020_0 := false;
   AI_RAW_7216.___________0020_1 := false;
   AI_RAW_7216.RAW_MIN := -2000;
   AI_RAW_7216.RAW_MAX := 8500;
   AI_RAW_7216.RAW_DESC := 'Thermal Resistance - 4-wire (Pt50 standard - 3902)';
   AI_RAW_7216.___________0030_1 := false;
   AI_RAW_7216.___________0030_2 := false;
   AI_RAW_7216.PARAM_TYPE := 16#07;
   AI_RAW_7216.PARAM_RANGE := 16#16;
   AI_RAW_7216.PARAM_COEF := 16#02;
   AI_RAW_7216.___________0040_1 := false;
   AI_RAW_7216.___________0040_2 := false;
   AI_RAW_7216.VALUE_COEF := 0.003902;
   AI_RAW_7516.revInfo.REV_BLOCK := 'UT00801';
   AI_RAW_7516.revInfo.REV_NUMBER := '001.000';
   AI_RAW_7516.revInfo.REV_DATE := '2024-04-09';
   AI_RAW_7516.revInfo.REV_AUTHOR := 'M. Gledhill';
   AI_RAW_7516.___________0010_0 := false;
   AI_RAW_7516.___________0010_1 := false;
   AI_RAW_7516.AI_CODE := 16#7516;
   AI_RAW_7516.___________0020_0 := false;
   AI_RAW_7516.___________0020_1 := false;
   AI_RAW_7516.RAW_MIN := -2000;
   AI_RAW_7516.RAW_MAX := 8500;
   AI_RAW_7516.RAW_DESC := 'Thermal Resistance - 4-wire (Pt50 standard - 391)';
   AI_RAW_7516.___________0030_1 := false;
   AI_RAW_7516.___________0030_2 := false;
   AI_RAW_7516.PARAM_TYPE := 16#07;
   AI_RAW_7516.PARAM_RANGE := 16#16;
   AI_RAW_7516.PARAM_COEF := 16#05;
   AI_RAW_7516.___________0040_1 := false;
   AI_RAW_7516.___________0040_2 := false;
   AI_RAW_7516.VALUE_COEF := 0.00391;
   AI_RAW_7116.revInfo.REV_BLOCK := 'UT00801';
   AI_RAW_7116.revInfo.REV_NUMBER := '001.000';
   AI_RAW_7116.revInfo.REV_DATE := '2024-04-09';
   AI_RAW_7116.revInfo.REV_AUTHOR := 'M. Gledhill';
   AI_RAW_7116.___________0010_0 := false;
   AI_RAW_7116.___________0010_1 := false;
   AI_RAW_7116.AI_CODE := 16#7116;
   AI_RAW_7116.___________0020_0 := false;
   AI_RAW_7116.___________0020_1 := false;
   AI_RAW_7116.RAW_MIN := -2000;
   AI_RAW_7116.RAW_MAX := 8500;
   AI_RAW_7116.RAW_DESC := 'Thermal Resistance - 4-wire (Pt50 standard - 3916)';
   AI_RAW_7116.___________0030_1 := false;
   AI_RAW_7116.___________0030_2 := false;
   AI_RAW_7116.PARAM_TYPE := 16#07;
   AI_RAW_7116.PARAM_RANGE := 16#16;
   AI_RAW_7116.PARAM_COEF := 16#01;
   AI_RAW_7116.___________0040_1 := false;
   AI_RAW_7116.___________0040_2 := false;
   AI_RAW_7116.VALUE_COEF := 0.003916;
   AI_RAW_7316.revInfo.REV_BLOCK := 'UT00801';
   AI_RAW_7316.revInfo.REV_NUMBER := '001.000';
   AI_RAW_7316.revInfo.REV_DATE := '2024-04-09';
   AI_RAW_7316.revInfo.REV_AUTHOR := 'M. Gledhill';
   AI_RAW_7316.___________0010_0 := false;
   AI_RAW_7316.___________0010_1 := false;
   AI_RAW_7316.AI_CODE := 16#7316;
   AI_RAW_7316.___________0020_0 := false;
   AI_RAW_7316.___________0020_1 := false;
   AI_RAW_7316.RAW_MIN := -2000;
   AI_RAW_7316.RAW_MAX := 8500;
   AI_RAW_7316.RAW_DESC := 'Thermal Resistance - 4-wire (Pt50 standard - 392)';
   AI_RAW_7316.___________0030_1 := false;
   AI_RAW_7316.___________0030_2 := false;
   AI_RAW_7316.PARAM_TYPE := 16#07;
   AI_RAW_7316.PARAM_RANGE := 16#16;
   AI_RAW_7316.PARAM_COEF := 16#03;
   AI_RAW_7316.___________0040_1 := false;
   AI_RAW_7316.___________0040_2 := false;
   AI_RAW_7316.VALUE_COEF := 0.00392;
   AI_RAW_7000.revInfo.REV_BLOCK := 'UT00801';
   AI_RAW_7000.revInfo.REV_NUMBER := '001.000';
   AI_RAW_7000.revInfo.REV_DATE := '2024-04-09';
   AI_RAW_7000.revInfo.REV_AUTHOR := 'M. Gledhill';
   AI_RAW_7000.___________0010_0 := false;
   AI_RAW_7000.___________0010_1 := false;
   AI_RAW_7000.AI_CODE := 16#7000;
   AI_RAW_7000.___________0020_0 := false;
   AI_RAW_7000.___________0020_1 := false;
   AI_RAW_7000.RAW_MIN := -12000;
   AI_RAW_7000.RAW_MAX := 13000;
   AI_RAW_7000.RAW_DESC := 'Thermal Resistance - 4-wire (Pt100 climate - 3851)';
   AI_RAW_7000.___________0030_1 := false;
   AI_RAW_7000.___________0030_2 := false;
   AI_RAW_7000.PARAM_TYPE := 16#07;
   AI_RAW_7000.PARAM_RANGE := 16#00;
   AI_RAW_7000.PARAM_COEF := 16#00;
   AI_RAW_7000.___________0040_1 := false;
   AI_RAW_7000.___________0040_2 := false;
   AI_RAW_7000.VALUE_COEF := 0.003851;
   AI_RAW_7200.revInfo.REV_BLOCK := 'UT00801';
   AI_RAW_7200.revInfo.REV_NUMBER := '001.000';
   AI_RAW_7200.revInfo.REV_DATE := '2024-04-09';
   AI_RAW_7200.revInfo.REV_AUTHOR := 'M. Gledhill';
   AI_RAW_7200.___________0010_0 := false;
   AI_RAW_7200.___________0010_1 := false;
   AI_RAW_7200.AI_CODE := 16#7200;
   AI_RAW_7200.___________0020_0 := false;
   AI_RAW_7200.___________0020_1 := false;
   AI_RAW_7200.RAW_MIN := -12000;
   AI_RAW_7200.RAW_MAX := 13000;
   AI_RAW_7200.RAW_DESC := 'Thermal Resistance - 4-wire (Pt100 climate - 3902)';
   AI_RAW_7200.___________0030_1 := false;
   AI_RAW_7200.___________0030_2 := false;
   AI_RAW_7200.PARAM_TYPE := 16#07;
   AI_RAW_7200.PARAM_RANGE := 16#00;
   AI_RAW_7200.PARAM_COEF := 16#02;
   AI_RAW_7200.___________0040_1 := false;
   AI_RAW_7200.___________0040_2 := false;
   AI_RAW_7200.VALUE_COEF := 0.003902;
   AI_RAW_7500.revInfo.REV_BLOCK := 'UT00801';
   AI_RAW_7500.revInfo.REV_NUMBER := '001.000';
   AI_RAW_7500.revInfo.REV_DATE := '2024-04-09';
   AI_RAW_7500.revInfo.REV_AUTHOR := 'M. Gledhill';
   AI_RAW_7500.___________0010_0 := false;
   AI_RAW_7500.___________0010_1 := false;
   AI_RAW_7500.AI_CODE := 16#7500;
   AI_RAW_7500.___________0020_0 := false;
   AI_RAW_7500.___________0020_1 := false;
   AI_RAW_7500.RAW_MIN := -12000;
   AI_RAW_7500.RAW_MAX := 13000;
   AI_RAW_7500.RAW_DESC := 'Thermal Resistance - 4-wire (Pt100 climate - 391)';
   AI_RAW_7500.___________0030_1 := false;
   AI_RAW_7500.___________0030_2 := false;
   AI_RAW_7500.PARAM_TYPE := 16#07;
   AI_RAW_7500.PARAM_RANGE := 16#00;
   AI_RAW_7500.PARAM_COEF := 16#05;
   AI_RAW_7500.___________0040_1 := false;
   AI_RAW_7500.___________0040_2 := false;
   AI_RAW_7500.VALUE_COEF := 0.00391;
   AI_RAW_7100.revInfo.REV_BLOCK := 'UT00801';
   AI_RAW_7100.revInfo.REV_NUMBER := '001.000';
   AI_RAW_7100.revInfo.REV_DATE := '2024-04-09';
   AI_RAW_7100.revInfo.REV_AUTHOR := 'M. Gledhill';
   AI_RAW_7100.___________0010_0 := false;
   AI_RAW_7100.___________0010_1 := false;
   AI_RAW_7100.AI_CODE := 16#7100;
   AI_RAW_7100.___________0020_0 := false;
   AI_RAW_7100.___________0020_1 := false;
   AI_RAW_7100.RAW_MIN := -12000;
   AI_RAW_7100.RAW_MAX := 13000;
   AI_RAW_7100.RAW_DESC := 'Thermal Resistance - 4-wire (Pt100 climate - 3916)';
   AI_RAW_7100.___________0030_1 := false;
   AI_RAW_7100.___________0030_2 := false;
   AI_RAW_7100.PARAM_TYPE := 16#07;
   AI_RAW_7100.PARAM_RANGE := 16#00;
   AI_RAW_7100.PARAM_COEF := 16#01;
   AI_RAW_7100.___________0040_1 := false;
   AI_RAW_7100.___________0040_2 := false;
   AI_RAW_7100.VALUE_COEF := 0.003916;
   AI_RAW_7300.revInfo.REV_BLOCK := 'UT00801';
   AI_RAW_7300.revInfo.REV_NUMBER := '001.000';
   AI_RAW_7300.revInfo.REV_DATE := '2024-04-09';
   AI_RAW_7300.revInfo.REV_AUTHOR := 'M. Gledhill';
   AI_RAW_7300.___________0010_0 := false;
   AI_RAW_7300.___________0010_1 := false;
   AI_RAW_7300.AI_CODE := 16#7300;
   AI_RAW_7300.___________0020_0 := false;
   AI_RAW_7300.___________0020_1 := false;
   AI_RAW_7300.RAW_MIN := -12000;
   AI_RAW_7300.RAW_MAX := 13000;
   AI_RAW_7300.RAW_DESC := 'Thermal Resistance - 4-wire (Pt100 climate - 392)';
   AI_RAW_7300.___________0030_1 := false;
   AI_RAW_7300.___________0030_2 := false;
   AI_RAW_7300.PARAM_TYPE := 16#07;
   AI_RAW_7300.PARAM_RANGE := 16#00;
   AI_RAW_7300.PARAM_COEF := 16#03;
   AI_RAW_7300.___________0040_1 := false;
   AI_RAW_7300.___________0040_2 := false;
   AI_RAW_7300.VALUE_COEF := 0.00392;
   AI_RAW_7002.revInfo.REV_BLOCK := 'UT00801';
   AI_RAW_7002.revInfo.REV_NUMBER := '001.000';
   AI_RAW_7002.revInfo.REV_DATE := '2024-04-09';
   AI_RAW_7002.revInfo.REV_AUTHOR := 'M. Gledhill';
   AI_RAW_7002.___________0010_0 := false;
   AI_RAW_7002.___________0010_1 := false;
   AI_RAW_7002.AI_CODE := 16#7002;
   AI_RAW_7002.___________0020_0 := false;
   AI_RAW_7002.___________0020_1 := false;
   AI_RAW_7002.RAW_MIN := -2000;
   AI_RAW_7002.RAW_MAX := 8500;
   AI_RAW_7002.RAW_DESC := 'Thermal Resistance - 4-wire (Pt100 standard - 3851)';
   AI_RAW_7002.___________0030_1 := false;
   AI_RAW_7002.___________0030_2 := false;
   AI_RAW_7002.PARAM_TYPE := 16#07;
   AI_RAW_7002.PARAM_RANGE := 16#02;
   AI_RAW_7002.PARAM_COEF := 16#00;
   AI_RAW_7002.___________0040_1 := false;
   AI_RAW_7002.___________0040_2 := false;
   AI_RAW_7002.VALUE_COEF := 0.003851;
   AI_RAW_7202.revInfo.REV_BLOCK := 'UT00801';
   AI_RAW_7202.revInfo.REV_NUMBER := '001.000';
   AI_RAW_7202.revInfo.REV_DATE := '2024-04-09';
   AI_RAW_7202.revInfo.REV_AUTHOR := 'M. Gledhill';
   AI_RAW_7202.___________0010_0 := false;
   AI_RAW_7202.___________0010_1 := false;
   AI_RAW_7202.AI_CODE := 16#7202;
   AI_RAW_7202.___________0020_0 := false;
   AI_RAW_7202.___________0020_1 := false;
   AI_RAW_7202.RAW_MIN := -2000;
   AI_RAW_7202.RAW_MAX := 8500;
   AI_RAW_7202.RAW_DESC := 'Thermal Resistance - 4-wire (Pt100 standard - 3902)';
   AI_RAW_7202.___________0030_1 := false;
   AI_RAW_7202.___________0030_2 := false;
   AI_RAW_7202.PARAM_TYPE := 16#07;
   AI_RAW_7202.PARAM_RANGE := 16#02;
   AI_RAW_7202.PARAM_COEF := 16#02;
   AI_RAW_7202.___________0040_1 := false;
   AI_RAW_7202.___________0040_2 := false;
   AI_RAW_7202.VALUE_COEF := 0.003902;
   AI_RAW_7502.revInfo.REV_BLOCK := 'UT00801';
   AI_RAW_7502.revInfo.REV_NUMBER := '001.000';
   AI_RAW_7502.revInfo.REV_DATE := '2024-04-09';
   AI_RAW_7502.revInfo.REV_AUTHOR := 'M. Gledhill';
   AI_RAW_7502.___________0010_0 := false;
   AI_RAW_7502.___________0010_1 := false;
   AI_RAW_7502.AI_CODE := 16#7502;
   AI_RAW_7502.___________0020_0 := false;
   AI_RAW_7502.___________0020_1 := false;
   AI_RAW_7502.RAW_MIN := -2000;
   AI_RAW_7502.RAW_MAX := 8500;
   AI_RAW_7502.RAW_DESC := 'Thermal Resistance - 4-wire (Pt100 standard - 391)';
   AI_RAW_7502.___________0030_1 := false;
   AI_RAW_7502.___________0030_2 := false;
   AI_RAW_7502.PARAM_TYPE := 16#07;
   AI_RAW_7502.PARAM_RANGE := 16#02;
   AI_RAW_7502.PARAM_COEF := 16#05;
   AI_RAW_7502.___________0040_1 := false;
   AI_RAW_7502.___________0040_2 := false;
   AI_RAW_7502.VALUE_COEF := 0.00391;
   AI_RAW_7102.revInfo.REV_BLOCK := 'UT00801';
   AI_RAW_7102.revInfo.REV_NUMBER := '001.000';
   AI_RAW_7102.revInfo.REV_DATE := '2024-04-09';
   AI_RAW_7102.revInfo.REV_AUTHOR := 'M. Gledhill';
   AI_RAW_7102.___________0010_0 := false;
   AI_RAW_7102.___________0010_1 := false;
   AI_RAW_7102.AI_CODE := 16#7102;
   AI_RAW_7102.___________0020_0 := false;
   AI_RAW_7102.___________0020_1 := false;
   AI_RAW_7102.RAW_MIN := -2000;
   AI_RAW_7102.RAW_MAX := 8500;
   AI_RAW_7102.RAW_DESC := 'Thermal Resistance - 4-wire (Pt100 standard - 3916)';
   AI_RAW_7102.___________0030_1 := false;
   AI_RAW_7102.___________0030_2 := false;
   AI_RAW_7102.PARAM_TYPE := 16#07;
   AI_RAW_7102.PARAM_RANGE := 16#02;
   AI_RAW_7102.PARAM_COEF := 16#01;
   AI_RAW_7102.___________0040_1 := false;
   AI_RAW_7102.___________0040_2 := false;
   AI_RAW_7102.VALUE_COEF := 0.003916;
   AI_RAW_7302.revInfo.REV_BLOCK := 'UT00801';
   AI_RAW_7302.revInfo.REV_NUMBER := '001.000';
   AI_RAW_7302.revInfo.REV_DATE := '2024-04-09';
   AI_RAW_7302.revInfo.REV_AUTHOR := 'M. Gledhill';
   AI_RAW_7302.___________0010_0 := false;
   AI_RAW_7302.___________0010_1 := false;
   AI_RAW_7302.AI_CODE := 16#7302;
   AI_RAW_7302.___________0020_0 := false;
   AI_RAW_7302.___________0020_1 := false;
   AI_RAW_7302.RAW_MIN := -2000;
   AI_RAW_7302.RAW_MAX := 8500;
   AI_RAW_7302.RAW_DESC := 'Thermal Resistance - 4-wire (Pt100 standard - 392)';
   AI_RAW_7302.___________0030_1 := false;
   AI_RAW_7302.___________0030_2 := false;
   AI_RAW_7302.PARAM_TYPE := 16#07;
   AI_RAW_7302.PARAM_RANGE := 16#02;
   AI_RAW_7302.PARAM_COEF := 16#03;
   AI_RAW_7302.___________0040_1 := false;
   AI_RAW_7302.___________0040_2 := false;
   AI_RAW_7302.VALUE_COEF := 0.00392;
   AI_RAW_7007.revInfo.REV_BLOCK := 'UT00801';
   AI_RAW_7007.revInfo.REV_NUMBER := '001.000';
   AI_RAW_7007.revInfo.REV_DATE := '2024-04-09';
   AI_RAW_7007.revInfo.REV_AUTHOR := 'M. Gledhill';
   AI_RAW_7007.___________0010_0 := false;
   AI_RAW_7007.___________0010_1 := false;
   AI_RAW_7007.AI_CODE := 16#7007;
   AI_RAW_7007.___________0020_0 := false;
   AI_RAW_7007.___________0020_1 := false;
   AI_RAW_7007.RAW_MIN := -12000;
   AI_RAW_7007.RAW_MAX := 13000;
   AI_RAW_7007.RAW_DESC := 'Thermal Resistance - 4-wire (Pt200 climate - 3851)';
   AI_RAW_7007.___________0030_1 := false;
   AI_RAW_7007.___________0030_2 := false;
   AI_RAW_7007.PARAM_TYPE := 16#07;
   AI_RAW_7007.PARAM_RANGE := 16#07;
   AI_RAW_7007.PARAM_COEF := 16#00;
   AI_RAW_7007.___________0040_1 := false;
   AI_RAW_7007.___________0040_2 := false;
   AI_RAW_7007.VALUE_COEF := 0.003851;
   AI_RAW_7207.revInfo.REV_BLOCK := 'UT00801';
   AI_RAW_7207.revInfo.REV_NUMBER := '001.000';
   AI_RAW_7207.revInfo.REV_DATE := '2024-04-09';
   AI_RAW_7207.revInfo.REV_AUTHOR := 'M. Gledhill';
   AI_RAW_7207.___________0010_0 := false;
   AI_RAW_7207.___________0010_1 := false;
   AI_RAW_7207.AI_CODE := 16#7207;
   AI_RAW_7207.___________0020_0 := false;
   AI_RAW_7207.___________0020_1 := false;
   AI_RAW_7207.RAW_MIN := -12000;
   AI_RAW_7207.RAW_MAX := 13000;
   AI_RAW_7207.RAW_DESC := 'Thermal Resistance - 4-wire (Pt200 climate - 3902)';
   AI_RAW_7207.___________0030_1 := false;
   AI_RAW_7207.___________0030_2 := false;
   AI_RAW_7207.PARAM_TYPE := 16#07;
   AI_RAW_7207.PARAM_RANGE := 16#07;
   AI_RAW_7207.PARAM_COEF := 16#02;
   AI_RAW_7207.___________0040_1 := false;
   AI_RAW_7207.___________0040_2 := false;
   AI_RAW_7207.VALUE_COEF := 0.003902;
   AI_RAW_7507.revInfo.REV_BLOCK := 'UT00801';
   AI_RAW_7507.revInfo.REV_NUMBER := '001.000';
   AI_RAW_7507.revInfo.REV_DATE := '2024-04-09';
   AI_RAW_7507.revInfo.REV_AUTHOR := 'M. Gledhill';
   AI_RAW_7507.___________0010_0 := false;
   AI_RAW_7507.___________0010_1 := false;
   AI_RAW_7507.AI_CODE := 16#7507;
   AI_RAW_7507.___________0020_0 := false;
   AI_RAW_7507.___________0020_1 := false;
   AI_RAW_7507.RAW_MIN := -12000;
   AI_RAW_7507.RAW_MAX := 13000;
   AI_RAW_7507.RAW_DESC := 'Thermal Resistance - 4-wire (Pt200 climate - 391)';
   AI_RAW_7507.___________0030_1 := false;
   AI_RAW_7507.___________0030_2 := false;
   AI_RAW_7507.PARAM_TYPE := 16#07;
   AI_RAW_7507.PARAM_RANGE := 16#07;
   AI_RAW_7507.PARAM_COEF := 16#05;
   AI_RAW_7507.___________0040_1 := false;
   AI_RAW_7507.___________0040_2 := false;
   AI_RAW_7507.VALUE_COEF := 0.00391;
   AI_RAW_7107.revInfo.REV_BLOCK := 'UT00801';
   AI_RAW_7107.revInfo.REV_NUMBER := '001.000';
   AI_RAW_7107.revInfo.REV_DATE := '2024-04-09';
   AI_RAW_7107.revInfo.REV_AUTHOR := 'M. Gledhill';
   AI_RAW_7107.___________0010_0 := false;
   AI_RAW_7107.___________0010_1 := false;
   AI_RAW_7107.AI_CODE := 16#7107;
   AI_RAW_7107.___________0020_0 := false;
   AI_RAW_7107.___________0020_1 := false;
   AI_RAW_7107.RAW_MIN := -12000;
   AI_RAW_7107.RAW_MAX := 13000;
   AI_RAW_7107.RAW_DESC := 'Thermal Resistance - 4-wire (Pt200 climate - 3916)';
   AI_RAW_7107.___________0030_1 := false;
   AI_RAW_7107.___________0030_2 := false;
   AI_RAW_7107.PARAM_TYPE := 16#07;
   AI_RAW_7107.PARAM_RANGE := 16#07;
   AI_RAW_7107.PARAM_COEF := 16#01;
   AI_RAW_7107.___________0040_1 := false;
   AI_RAW_7107.___________0040_2 := false;
   AI_RAW_7107.VALUE_COEF := 0.003916;
   AI_RAW_7307.revInfo.REV_BLOCK := 'UT00801';
   AI_RAW_7307.revInfo.REV_NUMBER := '001.000';
   AI_RAW_7307.revInfo.REV_DATE := '2024-04-09';
   AI_RAW_7307.revInfo.REV_AUTHOR := 'M. Gledhill';
   AI_RAW_7307.___________0010_0 := false;
   AI_RAW_7307.___________0010_1 := false;
   AI_RAW_7307.AI_CODE := 16#7307;
   AI_RAW_7307.___________0020_0 := false;
   AI_RAW_7307.___________0020_1 := false;
   AI_RAW_7307.RAW_MIN := -12000;
   AI_RAW_7307.RAW_MAX := 13000;
   AI_RAW_7307.RAW_DESC := 'Thermal Resistance - 4-wire (Pt200 climate - 392)';
   AI_RAW_7307.___________0030_1 := false;
   AI_RAW_7307.___________0030_2 := false;
   AI_RAW_7307.PARAM_TYPE := 16#07;
   AI_RAW_7307.PARAM_RANGE := 16#07;
   AI_RAW_7307.PARAM_COEF := 16#03;
   AI_RAW_7307.___________0040_1 := false;
   AI_RAW_7307.___________0040_2 := false;
   AI_RAW_7307.VALUE_COEF := 0.00392;
   AI_RAW_700B.revInfo.REV_BLOCK := 'UT00801';
   AI_RAW_700B.revInfo.REV_NUMBER := '001.000';
   AI_RAW_700B.revInfo.REV_DATE := '2024-04-09';
   AI_RAW_700B.revInfo.REV_AUTHOR := 'M. Gledhill';
   AI_RAW_700B.___________0010_0 := false;
   AI_RAW_700B.___________0010_1 := false;
   AI_RAW_700B.AI_CODE := 16#700B;
   AI_RAW_700B.___________0020_0 := false;
   AI_RAW_700B.___________0020_1 := false;
   AI_RAW_700B.RAW_MIN := -2000;
   AI_RAW_700B.RAW_MAX := 8500;
   AI_RAW_700B.RAW_DESC := 'Thermal Resistance - 4-wire (Pt200 standard - 3851)';
   AI_RAW_700B.___________0030_1 := false;
   AI_RAW_700B.___________0030_2 := false;
   AI_RAW_700B.PARAM_TYPE := 16#07;
   AI_RAW_700B.PARAM_RANGE := 16#0B;
   AI_RAW_700B.PARAM_COEF := 16#00;
   AI_RAW_700B.___________0040_1 := false;
   AI_RAW_700B.___________0040_2 := false;
   AI_RAW_700B.VALUE_COEF := 0.003851;
   AI_RAW_720B.revInfo.REV_BLOCK := 'UT00801';
   AI_RAW_720B.revInfo.REV_NUMBER := '001.000';
   AI_RAW_720B.revInfo.REV_DATE := '2024-04-09';
   AI_RAW_720B.revInfo.REV_AUTHOR := 'M. Gledhill';
   AI_RAW_720B.___________0010_0 := false;
   AI_RAW_720B.___________0010_1 := false;
   AI_RAW_720B.AI_CODE := 16#720B;
   AI_RAW_720B.___________0020_0 := false;
   AI_RAW_720B.___________0020_1 := false;
   AI_RAW_720B.RAW_MIN := -2000;
   AI_RAW_720B.RAW_MAX := 8500;
   AI_RAW_720B.RAW_DESC := 'Thermal Resistance - 4-wire (Pt200 standard - 3902)';
   AI_RAW_720B.___________0030_1 := false;
   AI_RAW_720B.___________0030_2 := false;
   AI_RAW_720B.PARAM_TYPE := 16#07;
   AI_RAW_720B.PARAM_RANGE := 16#0B;
   AI_RAW_720B.PARAM_COEF := 16#02;
   AI_RAW_720B.___________0040_1 := false;
   AI_RAW_720B.___________0040_2 := false;
   AI_RAW_720B.VALUE_COEF := 0.003902;
   AI_RAW_750B.revInfo.REV_BLOCK := 'UT00801';
   AI_RAW_750B.revInfo.REV_NUMBER := '001.000';
   AI_RAW_750B.revInfo.REV_DATE := '2024-04-09';
   AI_RAW_750B.revInfo.REV_AUTHOR := 'M. Gledhill';
   AI_RAW_750B.___________0010_0 := false;
   AI_RAW_750B.___________0010_1 := false;
   AI_RAW_750B.AI_CODE := 16#750B;
   AI_RAW_750B.___________0020_0 := false;
   AI_RAW_750B.___________0020_1 := false;
   AI_RAW_750B.RAW_MIN := -2000;
   AI_RAW_750B.RAW_MAX := 8500;
   AI_RAW_750B.RAW_DESC := 'Thermal Resistance - 4-wire (Pt200 standard - 391)';
   AI_RAW_750B.___________0030_1 := false;
   AI_RAW_750B.___________0030_2 := false;
   AI_RAW_750B.PARAM_TYPE := 16#07;
   AI_RAW_750B.PARAM_RANGE := 16#0B;
   AI_RAW_750B.PARAM_COEF := 16#05;
   AI_RAW_750B.___________0040_1 := false;
   AI_RAW_750B.___________0040_2 := false;
   AI_RAW_750B.VALUE_COEF := 0.00391;
   AI_RAW_710B.revInfo.REV_BLOCK := 'UT00801';
   AI_RAW_710B.revInfo.REV_NUMBER := '001.000';
   AI_RAW_710B.revInfo.REV_DATE := '2024-04-09';
   AI_RAW_710B.revInfo.REV_AUTHOR := 'M. Gledhill';
   AI_RAW_710B.___________0010_0 := false;
   AI_RAW_710B.___________0010_1 := false;
   AI_RAW_710B.AI_CODE := 16#710B;
   AI_RAW_710B.___________0020_0 := false;
   AI_RAW_710B.___________0020_1 := false;
   AI_RAW_710B.RAW_MIN := -2000;
   AI_RAW_710B.RAW_MAX := 8500;
   AI_RAW_710B.RAW_DESC := 'Thermal Resistance - 4-wire (Pt200 standard - 3916)';
   AI_RAW_710B.___________0030_1 := false;
   AI_RAW_710B.___________0030_2 := false;
   AI_RAW_710B.PARAM_TYPE := 16#07;
   AI_RAW_710B.PARAM_RANGE := 16#0B;
   AI_RAW_710B.PARAM_COEF := 16#01;
   AI_RAW_710B.___________0040_1 := false;
   AI_RAW_710B.___________0040_2 := false;
   AI_RAW_710B.VALUE_COEF := 0.003916;
   AI_RAW_730B.revInfo.REV_BLOCK := 'UT00801';
   AI_RAW_730B.revInfo.REV_NUMBER := '001.000';
   AI_RAW_730B.revInfo.REV_DATE := '2024-04-09';
   AI_RAW_730B.revInfo.REV_AUTHOR := 'M. Gledhill';
   AI_RAW_730B.___________0010_0 := false;
   AI_RAW_730B.___________0010_1 := false;
   AI_RAW_730B.AI_CODE := 16#730B;
   AI_RAW_730B.___________0020_0 := false;
   AI_RAW_730B.___________0020_1 := false;
   AI_RAW_730B.RAW_MIN := -2000;
   AI_RAW_730B.RAW_MAX := 8500;
   AI_RAW_730B.RAW_DESC := 'Thermal Resistance - 4-wire (Pt200 standard - 392)';
   AI_RAW_730B.___________0030_1 := false;
   AI_RAW_730B.___________0030_2 := false;
   AI_RAW_730B.PARAM_TYPE := 16#07;
   AI_RAW_730B.PARAM_RANGE := 16#0B;
   AI_RAW_730B.PARAM_COEF := 16#03;
   AI_RAW_730B.___________0040_1 := false;
   AI_RAW_730B.___________0040_2 := false;
   AI_RAW_730B.VALUE_COEF := 0.00392;
   AI_RAW_7008.revInfo.REV_BLOCK := 'UT00801';
   AI_RAW_7008.revInfo.REV_NUMBER := '001.000';
   AI_RAW_7008.revInfo.REV_DATE := '2024-04-09';
   AI_RAW_7008.revInfo.REV_AUTHOR := 'M. Gledhill';
   AI_RAW_7008.___________0010_0 := false;
   AI_RAW_7008.___________0010_1 := false;
   AI_RAW_7008.AI_CODE := 16#7008;
   AI_RAW_7008.___________0020_0 := false;
   AI_RAW_7008.___________0020_1 := false;
   AI_RAW_7008.RAW_MIN := -12000;
   AI_RAW_7008.RAW_MAX := 13000;
   AI_RAW_7008.RAW_DESC := 'Thermal Resistance - 4-wire (Pt500 climate - 3851)';
   AI_RAW_7008.___________0030_1 := false;
   AI_RAW_7008.___________0030_2 := false;
   AI_RAW_7008.PARAM_TYPE := 16#07;
   AI_RAW_7008.PARAM_RANGE := 16#08;
   AI_RAW_7008.PARAM_COEF := 16#00;
   AI_RAW_7008.___________0040_1 := false;
   AI_RAW_7008.___________0040_2 := false;
   AI_RAW_7008.VALUE_COEF := 0.003851;
   AI_RAW_7208.revInfo.REV_BLOCK := 'UT00801';
   AI_RAW_7208.revInfo.REV_NUMBER := '001.000';
   AI_RAW_7208.revInfo.REV_DATE := '2024-04-09';
   AI_RAW_7208.revInfo.REV_AUTHOR := 'M. Gledhill';
   AI_RAW_7208.___________0010_0 := false;
   AI_RAW_7208.___________0010_1 := false;
   AI_RAW_7208.AI_CODE := 16#7208;
   AI_RAW_7208.___________0020_0 := false;
   AI_RAW_7208.___________0020_1 := false;
   AI_RAW_7208.RAW_MIN := -12000;
   AI_RAW_7208.RAW_MAX := 13000;
   AI_RAW_7208.RAW_DESC := 'Thermal Resistance - 4-wire (Pt500 climate - 3902)';
   AI_RAW_7208.___________0030_1 := false;
   AI_RAW_7208.___________0030_2 := false;
   AI_RAW_7208.PARAM_TYPE := 16#07;
   AI_RAW_7208.PARAM_RANGE := 16#08;
   AI_RAW_7208.PARAM_COEF := 16#02;
   AI_RAW_7208.___________0040_1 := false;
   AI_RAW_7208.___________0040_2 := false;
   AI_RAW_7208.VALUE_COEF := 0.003902;
   AI_RAW_7508.revInfo.REV_BLOCK := 'UT00801';
   AI_RAW_7508.revInfo.REV_NUMBER := '001.000';
   AI_RAW_7508.revInfo.REV_DATE := '2024-04-09';
   AI_RAW_7508.revInfo.REV_AUTHOR := 'M. Gledhill';
   AI_RAW_7508.___________0010_0 := false;
   AI_RAW_7508.___________0010_1 := false;
   AI_RAW_7508.AI_CODE := 16#7508;
   AI_RAW_7508.___________0020_0 := false;
   AI_RAW_7508.___________0020_1 := false;
   AI_RAW_7508.RAW_MIN := -12000;
   AI_RAW_7508.RAW_MAX := 13000;
   AI_RAW_7508.RAW_DESC := 'Thermal Resistance - 4-wire (Pt500 climate - 391)';
   AI_RAW_7508.___________0030_1 := false;
   AI_RAW_7508.___________0030_2 := false;
   AI_RAW_7508.PARAM_TYPE := 16#07;
   AI_RAW_7508.PARAM_RANGE := 16#08;
   AI_RAW_7508.PARAM_COEF := 16#05;
   AI_RAW_7508.___________0040_1 := false;
   AI_RAW_7508.___________0040_2 := false;
   AI_RAW_7508.VALUE_COEF := 0.00391;
   AI_RAW_7108.revInfo.REV_BLOCK := 'UT00801';
   AI_RAW_7108.revInfo.REV_NUMBER := '001.000';
   AI_RAW_7108.revInfo.REV_DATE := '2024-04-09';
   AI_RAW_7108.revInfo.REV_AUTHOR := 'M. Gledhill';
   AI_RAW_7108.___________0010_0 := false;
   AI_RAW_7108.___________0010_1 := false;
   AI_RAW_7108.AI_CODE := 16#7108;
   AI_RAW_7108.___________0020_0 := false;
   AI_RAW_7108.___________0020_1 := false;
   AI_RAW_7108.RAW_MIN := -12000;
   AI_RAW_7108.RAW_MAX := 13000;
   AI_RAW_7108.RAW_DESC := 'Thermal Resistance - 4-wire (Pt500 climate - 3916)';
   AI_RAW_7108.___________0030_1 := false;
   AI_RAW_7108.___________0030_2 := false;
   AI_RAW_7108.PARAM_TYPE := 16#07;
   AI_RAW_7108.PARAM_RANGE := 16#08;
   AI_RAW_7108.PARAM_COEF := 16#01;
   AI_RAW_7108.___________0040_1 := false;
   AI_RAW_7108.___________0040_2 := false;
   AI_RAW_7108.VALUE_COEF := 0.003916;
   AI_RAW_7308.revInfo.REV_BLOCK := 'UT00801';
   AI_RAW_7308.revInfo.REV_NUMBER := '001.000';
   AI_RAW_7308.revInfo.REV_DATE := '2024-04-09';
   AI_RAW_7308.revInfo.REV_AUTHOR := 'M. Gledhill';
   AI_RAW_7308.___________0010_0 := false;
   AI_RAW_7308.___________0010_1 := false;
   AI_RAW_7308.AI_CODE := 16#7308;
   AI_RAW_7308.___________0020_0 := false;
   AI_RAW_7308.___________0020_1 := false;
   AI_RAW_7308.RAW_MIN := -12000;
   AI_RAW_7308.RAW_MAX := 13000;
   AI_RAW_7308.RAW_DESC := 'Thermal Resistance - 4-wire (Pt500 climate - 392)';
   AI_RAW_7308.___________0030_1 := false;
   AI_RAW_7308.___________0030_2 := false;
   AI_RAW_7308.PARAM_TYPE := 16#07;
   AI_RAW_7308.PARAM_RANGE := 16#08;
   AI_RAW_7308.PARAM_COEF := 16#03;
   AI_RAW_7308.___________0040_1 := false;
   AI_RAW_7308.___________0040_2 := false;
   AI_RAW_7308.VALUE_COEF := 0.00392;
   AI_RAW_7004.revInfo.REV_BLOCK := 'UT00801';
   AI_RAW_7004.revInfo.REV_NUMBER := '001.000';
   AI_RAW_7004.revInfo.REV_DATE := '2024-04-09';
   AI_RAW_7004.revInfo.REV_AUTHOR := 'M. Gledhill';
   AI_RAW_7004.___________0010_0 := false;
   AI_RAW_7004.___________0010_1 := false;
   AI_RAW_7004.AI_CODE := 16#7004;
   AI_RAW_7004.___________0020_0 := false;
   AI_RAW_7004.___________0020_1 := false;
   AI_RAW_7004.RAW_MIN := -2000;
   AI_RAW_7004.RAW_MAX := 8500;
   AI_RAW_7004.RAW_DESC := 'Thermal Resistance - 4-wire (Pt500 standard - 3851)';
   AI_RAW_7004.___________0030_1 := false;
   AI_RAW_7004.___________0030_2 := false;
   AI_RAW_7004.PARAM_TYPE := 16#07;
   AI_RAW_7004.PARAM_RANGE := 16#04;
   AI_RAW_7004.PARAM_COEF := 16#00;
   AI_RAW_7004.___________0040_1 := false;
   AI_RAW_7004.___________0040_2 := false;
   AI_RAW_7004.VALUE_COEF := 0.003851;
   AI_RAW_7204.revInfo.REV_BLOCK := 'UT00801';
   AI_RAW_7204.revInfo.REV_NUMBER := '001.000';
   AI_RAW_7204.revInfo.REV_DATE := '2024-04-09';
   AI_RAW_7204.revInfo.REV_AUTHOR := 'M. Gledhill';
   AI_RAW_7204.___________0010_0 := false;
   AI_RAW_7204.___________0010_1 := false;
   AI_RAW_7204.AI_CODE := 16#7204;
   AI_RAW_7204.___________0020_0 := false;
   AI_RAW_7204.___________0020_1 := false;
   AI_RAW_7204.RAW_MIN := -2000;
   AI_RAW_7204.RAW_MAX := 8500;
   AI_RAW_7204.RAW_DESC := 'Thermal Resistance - 4-wire (Pt500 standard - 3902)';
   AI_RAW_7204.___________0030_1 := false;
   AI_RAW_7204.___________0030_2 := false;
   AI_RAW_7204.PARAM_TYPE := 16#07;
   AI_RAW_7204.PARAM_RANGE := 16#04;
   AI_RAW_7204.PARAM_COEF := 16#02;
   AI_RAW_7204.___________0040_1 := false;
   AI_RAW_7204.___________0040_2 := false;
   AI_RAW_7204.VALUE_COEF := 0.003902;
   AI_RAW_7504.revInfo.REV_BLOCK := 'UT00801';
   AI_RAW_7504.revInfo.REV_NUMBER := '001.000';
   AI_RAW_7504.revInfo.REV_DATE := '2024-04-09';
   AI_RAW_7504.revInfo.REV_AUTHOR := 'M. Gledhill';
   AI_RAW_7504.___________0010_0 := false;
   AI_RAW_7504.___________0010_1 := false;
   AI_RAW_7504.AI_CODE := 16#7504;
   AI_RAW_7504.___________0020_0 := false;
   AI_RAW_7504.___________0020_1 := false;
   AI_RAW_7504.RAW_MIN := -2000;
   AI_RAW_7504.RAW_MAX := 8500;
   AI_RAW_7504.RAW_DESC := 'Thermal Resistance - 4-wire (Pt500 standard - 391)';
   AI_RAW_7504.___________0030_1 := false;
   AI_RAW_7504.___________0030_2 := false;
   AI_RAW_7504.PARAM_TYPE := 16#07;
   AI_RAW_7504.PARAM_RANGE := 16#04;
   AI_RAW_7504.PARAM_COEF := 16#05;
   AI_RAW_7504.___________0040_1 := false;
   AI_RAW_7504.___________0040_2 := false;
   AI_RAW_7504.VALUE_COEF := 0.00391;
   AI_RAW_7104.revInfo.REV_BLOCK := 'UT00801';
   AI_RAW_7104.revInfo.REV_NUMBER := '001.000';
   AI_RAW_7104.revInfo.REV_DATE := '2024-04-09';
   AI_RAW_7104.revInfo.REV_AUTHOR := 'M. Gledhill';
   AI_RAW_7104.___________0010_0 := false;
   AI_RAW_7104.___________0010_1 := false;
   AI_RAW_7104.AI_CODE := 16#7104;
   AI_RAW_7104.___________0020_0 := false;
   AI_RAW_7104.___________0020_1 := false;
   AI_RAW_7104.RAW_MIN := -2000;
   AI_RAW_7104.RAW_MAX := 8500;
   AI_RAW_7104.RAW_DESC := 'Thermal Resistance - 4-wire (Pt500 standard - 3916)';
   AI_RAW_7104.___________0030_1 := false;
   AI_RAW_7104.___________0030_2 := false;
   AI_RAW_7104.PARAM_TYPE := 16#07;
   AI_RAW_7104.PARAM_RANGE := 16#04;
   AI_RAW_7104.PARAM_COEF := 16#01;
   AI_RAW_7104.___________0040_1 := false;
   AI_RAW_7104.___________0040_2 := false;
   AI_RAW_7104.VALUE_COEF := 0.003916;
   AI_RAW_7304.revInfo.REV_BLOCK := 'UT00801';
   AI_RAW_7304.revInfo.REV_NUMBER := '001.000';
   AI_RAW_7304.revInfo.REV_DATE := '2024-04-09';
   AI_RAW_7304.revInfo.REV_AUTHOR := 'M. Gledhill';
   AI_RAW_7304.___________0010_0 := false;
   AI_RAW_7304.___________0010_1 := false;
   AI_RAW_7304.AI_CODE := 16#7304;
   AI_RAW_7304.___________0020_0 := false;
   AI_RAW_7304.___________0020_1 := false;
   AI_RAW_7304.RAW_MIN := -2000;
   AI_RAW_7304.RAW_MAX := 8500;
   AI_RAW_7304.RAW_DESC := 'Thermal Resistance - 4-wire (Pt500 standard - 392)';
   AI_RAW_7304.___________0030_1 := false;
   AI_RAW_7304.___________0030_2 := false;
   AI_RAW_7304.PARAM_TYPE := 16#07;
   AI_RAW_7304.PARAM_RANGE := 16#04;
   AI_RAW_7304.PARAM_COEF := 16#03;
   AI_RAW_7304.___________0040_1 := false;
   AI_RAW_7304.___________0040_2 := false;
   AI_RAW_7304.VALUE_COEF := 0.00392;
   AI_RAW_7009.revInfo.REV_BLOCK := 'UT00801';
   AI_RAW_7009.revInfo.REV_NUMBER := '001.000';
   AI_RAW_7009.revInfo.REV_DATE := '2024-04-09';
   AI_RAW_7009.revInfo.REV_AUTHOR := 'M. Gledhill';
   AI_RAW_7009.___________0010_0 := false;
   AI_RAW_7009.___________0010_1 := false;
   AI_RAW_7009.AI_CODE := 16#7009;
   AI_RAW_7009.___________0020_0 := false;
   AI_RAW_7009.___________0020_1 := false;
   AI_RAW_7009.RAW_MIN := -12000;
   AI_RAW_7009.RAW_MAX := 13000;
   AI_RAW_7009.RAW_DESC := 'Thermal Resistance - 4-wire (Pt1000 climate - 3851)';
   AI_RAW_7009.___________0030_1 := false;
   AI_RAW_7009.___________0030_2 := false;
   AI_RAW_7009.PARAM_TYPE := 16#07;
   AI_RAW_7009.PARAM_RANGE := 16#09;
   AI_RAW_7009.PARAM_COEF := 16#00;
   AI_RAW_7009.___________0040_1 := false;
   AI_RAW_7009.___________0040_2 := false;
   AI_RAW_7009.VALUE_COEF := 0.003851;
   AI_RAW_7209.revInfo.REV_BLOCK := 'UT00801';
   AI_RAW_7209.revInfo.REV_NUMBER := '001.000';
   AI_RAW_7209.revInfo.REV_DATE := '2024-04-09';
   AI_RAW_7209.revInfo.REV_AUTHOR := 'M. Gledhill';
   AI_RAW_7209.___________0010_0 := false;
   AI_RAW_7209.___________0010_1 := false;
   AI_RAW_7209.AI_CODE := 16#7209;
   AI_RAW_7209.___________0020_0 := false;
   AI_RAW_7209.___________0020_1 := false;
   AI_RAW_7209.RAW_MIN := -12000;
   AI_RAW_7209.RAW_MAX := 13000;
   AI_RAW_7209.RAW_DESC := 'Thermal Resistance - 4-wire (Pt1000 climate - 3902)';
   AI_RAW_7209.___________0030_1 := false;
   AI_RAW_7209.___________0030_2 := false;
   AI_RAW_7209.PARAM_TYPE := 16#07;
   AI_RAW_7209.PARAM_RANGE := 16#09;
   AI_RAW_7209.PARAM_COEF := 16#02;
   AI_RAW_7209.___________0040_1 := false;
   AI_RAW_7209.___________0040_2 := false;
   AI_RAW_7209.VALUE_COEF := 0.003902;
   AI_RAW_7509.revInfo.REV_BLOCK := 'UT00801';
   AI_RAW_7509.revInfo.REV_NUMBER := '001.000';
   AI_RAW_7509.revInfo.REV_DATE := '2024-04-09';
   AI_RAW_7509.revInfo.REV_AUTHOR := 'M. Gledhill';
   AI_RAW_7509.___________0010_0 := false;
   AI_RAW_7509.___________0010_1 := false;
   AI_RAW_7509.AI_CODE := 16#7509;
   AI_RAW_7509.___________0020_0 := false;
   AI_RAW_7509.___________0020_1 := false;
   AI_RAW_7509.RAW_MIN := -12000;
   AI_RAW_7509.RAW_MAX := 13000;
   AI_RAW_7509.RAW_DESC := 'Thermal Resistance - 4-wire (Pt1000 climate - 391)';
   AI_RAW_7509.___________0030_1 := false;
   AI_RAW_7509.___________0030_2 := false;
   AI_RAW_7509.PARAM_TYPE := 16#07;
   AI_RAW_7509.PARAM_RANGE := 16#09;
   AI_RAW_7509.PARAM_COEF := 16#05;
   AI_RAW_7509.___________0040_1 := false;
   AI_RAW_7509.___________0040_2 := false;
   AI_RAW_7509.VALUE_COEF := 0.00391;
   AI_RAW_7109.revInfo.REV_BLOCK := 'UT00801';
   AI_RAW_7109.revInfo.REV_NUMBER := '001.000';
   AI_RAW_7109.revInfo.REV_DATE := '2024-04-09';
   AI_RAW_7109.revInfo.REV_AUTHOR := 'M. Gledhill';
   AI_RAW_7109.___________0010_0 := false;
   AI_RAW_7109.___________0010_1 := false;
   AI_RAW_7109.AI_CODE := 16#7109;
   AI_RAW_7109.___________0020_0 := false;
   AI_RAW_7109.___________0020_1 := false;
   AI_RAW_7109.RAW_MIN := -12000;
   AI_RAW_7109.RAW_MAX := 13000;
   AI_RAW_7109.RAW_DESC := 'Thermal Resistance - 4-wire (Pt1000 climate - 3916)';
   AI_RAW_7109.___________0030_1 := false;
   AI_RAW_7109.___________0030_2 := false;
   AI_RAW_7109.PARAM_TYPE := 16#07;
   AI_RAW_7109.PARAM_RANGE := 16#09;
   AI_RAW_7109.PARAM_COEF := 16#01;
   AI_RAW_7109.___________0040_1 := false;
   AI_RAW_7109.___________0040_2 := false;
   AI_RAW_7109.VALUE_COEF := 0.003916;
   AI_RAW_7309.revInfo.REV_BLOCK := 'UT00801';
   AI_RAW_7309.revInfo.REV_NUMBER := '001.000';
   AI_RAW_7309.revInfo.REV_DATE := '2024-04-09';
   AI_RAW_7309.revInfo.REV_AUTHOR := 'M. Gledhill';
   AI_RAW_7309.___________0010_0 := false;
   AI_RAW_7309.___________0010_1 := false;
   AI_RAW_7309.AI_CODE := 16#7309;
   AI_RAW_7309.___________0020_0 := false;
   AI_RAW_7309.___________0020_1 := false;
   AI_RAW_7309.RAW_MIN := -12000;
   AI_RAW_7309.RAW_MAX := 13000;
   AI_RAW_7309.RAW_DESC := 'Thermal Resistance - 4-wire (Pt1000 climate - 392)';
   AI_RAW_7309.___________0030_1 := false;
   AI_RAW_7309.___________0030_2 := false;
   AI_RAW_7309.PARAM_TYPE := 16#07;
   AI_RAW_7309.PARAM_RANGE := 16#09;
   AI_RAW_7309.PARAM_COEF := 16#03;
   AI_RAW_7309.___________0040_1 := false;
   AI_RAW_7309.___________0040_2 := false;
   AI_RAW_7309.VALUE_COEF := 0.00392;
   AI_RAW_7005.revInfo.REV_BLOCK := 'UT00801';
   AI_RAW_7005.revInfo.REV_NUMBER := '001.000';
   AI_RAW_7005.revInfo.REV_DATE := '2024-04-09';
   AI_RAW_7005.revInfo.REV_AUTHOR := 'M. Gledhill';
   AI_RAW_7005.___________0010_0 := false;
   AI_RAW_7005.___________0010_1 := false;
   AI_RAW_7005.AI_CODE := 16#7005;
   AI_RAW_7005.___________0020_0 := false;
   AI_RAW_7005.___________0020_1 := false;
   AI_RAW_7005.RAW_MIN := -2000;
   AI_RAW_7005.RAW_MAX := 8500;
   AI_RAW_7005.RAW_DESC := 'Thermal Resistance - 4-wire (Pt1000 standard - 3851)';
   AI_RAW_7005.___________0030_1 := false;
   AI_RAW_7005.___________0030_2 := false;
   AI_RAW_7005.PARAM_TYPE := 16#07;
   AI_RAW_7005.PARAM_RANGE := 16#05;
   AI_RAW_7005.PARAM_COEF := 16#00;
   AI_RAW_7005.___________0040_1 := false;
   AI_RAW_7005.___________0040_2 := false;
   AI_RAW_7005.VALUE_COEF := 0.003851;
   AI_RAW_7205.revInfo.REV_BLOCK := 'UT00801';
   AI_RAW_7205.revInfo.REV_NUMBER := '001.000';
   AI_RAW_7205.revInfo.REV_DATE := '2024-04-09';
   AI_RAW_7205.revInfo.REV_AUTHOR := 'M. Gledhill';
   AI_RAW_7205.___________0010_0 := false;
   AI_RAW_7205.___________0010_1 := false;
   AI_RAW_7205.AI_CODE := 16#7205;
   AI_RAW_7205.___________0020_0 := false;
   AI_RAW_7205.___________0020_1 := false;
   AI_RAW_7205.RAW_MIN := -2000;
   AI_RAW_7205.RAW_MAX := 8500;
   AI_RAW_7205.RAW_DESC := 'Thermal Resistance - 4-wire (Pt1000 standard - 3902)';
   AI_RAW_7205.___________0030_1 := false;
   AI_RAW_7205.___________0030_2 := false;
   AI_RAW_7205.PARAM_TYPE := 16#07;
   AI_RAW_7205.PARAM_RANGE := 16#05;
   AI_RAW_7205.PARAM_COEF := 16#02;
   AI_RAW_7205.___________0040_1 := false;
   AI_RAW_7205.___________0040_2 := false;
   AI_RAW_7205.VALUE_COEF := 0.003902;
   AI_RAW_7505.revInfo.REV_BLOCK := 'UT00801';
   AI_RAW_7505.revInfo.REV_NUMBER := '001.000';
   AI_RAW_7505.revInfo.REV_DATE := '2024-04-09';
   AI_RAW_7505.revInfo.REV_AUTHOR := 'M. Gledhill';
   AI_RAW_7505.___________0010_0 := false;
   AI_RAW_7505.___________0010_1 := false;
   AI_RAW_7505.AI_CODE := 16#7505;
   AI_RAW_7505.___________0020_0 := false;
   AI_RAW_7505.___________0020_1 := false;
   AI_RAW_7505.RAW_MIN := -2000;
   AI_RAW_7505.RAW_MAX := 8500;
   AI_RAW_7505.RAW_DESC := 'Thermal Resistance - 4-wire (Pt1000 standard - 391)';
   AI_RAW_7505.___________0030_1 := false;
   AI_RAW_7505.___________0030_2 := false;
   AI_RAW_7505.PARAM_TYPE := 16#07;
   AI_RAW_7505.PARAM_RANGE := 16#05;
   AI_RAW_7505.PARAM_COEF := 16#05;
   AI_RAW_7505.___________0040_1 := false;
   AI_RAW_7505.___________0040_2 := false;
   AI_RAW_7505.VALUE_COEF := 0.00391;
   AI_RAW_7105.revInfo.REV_BLOCK := 'UT00801';
   AI_RAW_7105.revInfo.REV_NUMBER := '001.000';
   AI_RAW_7105.revInfo.REV_DATE := '2024-04-09';
   AI_RAW_7105.revInfo.REV_AUTHOR := 'M. Gledhill';
   AI_RAW_7105.___________0010_0 := false;
   AI_RAW_7105.___________0010_1 := false;
   AI_RAW_7105.AI_CODE := 16#7105;
   AI_RAW_7105.___________0020_0 := false;
   AI_RAW_7105.___________0020_1 := false;
   AI_RAW_7105.RAW_MIN := -2000;
   AI_RAW_7105.RAW_MAX := 8500;
   AI_RAW_7105.RAW_DESC := 'Thermal Resistance - 4-wire (Pt1000 standard - 3916)';
   AI_RAW_7105.___________0030_1 := false;
   AI_RAW_7105.___________0030_2 := false;
   AI_RAW_7105.PARAM_TYPE := 16#07;
   AI_RAW_7105.PARAM_RANGE := 16#05;
   AI_RAW_7105.PARAM_COEF := 16#01;
   AI_RAW_7105.___________0040_1 := false;
   AI_RAW_7105.___________0040_2 := false;
   AI_RAW_7105.VALUE_COEF := 0.003916;
   AI_RAW_7305.revInfo.REV_BLOCK := 'UT00801';
   AI_RAW_7305.revInfo.REV_NUMBER := '001.000';
   AI_RAW_7305.revInfo.REV_DATE := '2024-04-09';
   AI_RAW_7305.revInfo.REV_AUTHOR := 'M. Gledhill';
   AI_RAW_7305.___________0010_0 := false;
   AI_RAW_7305.___________0010_1 := false;
   AI_RAW_7305.AI_CODE := 16#7305;
   AI_RAW_7305.___________0020_0 := false;
   AI_RAW_7305.___________0020_1 := false;
   AI_RAW_7305.RAW_MIN := -2000;
   AI_RAW_7305.RAW_MAX := 8500;
   AI_RAW_7305.RAW_DESC := 'Thermal Resistance - 4-wire (Pt1000 standard - 392)';
   AI_RAW_7305.___________0030_1 := false;
   AI_RAW_7305.___________0030_2 := false;
   AI_RAW_7305.PARAM_TYPE := 16#07;
   AI_RAW_7305.PARAM_RANGE := 16#05;
   AI_RAW_7305.PARAM_COEF := 16#03;
   AI_RAW_7305.___________0040_1 := false;
   AI_RAW_7305.___________0040_2 := false;
   AI_RAW_7305.VALUE_COEF := 0.00392;
   AI_RAW_8B0E.revInfo.REV_BLOCK := 'UT00801';
   AI_RAW_8B0E.revInfo.REV_NUMBER := '001.000';
   AI_RAW_8B0E.revInfo.REV_DATE := '2024-04-09';
   AI_RAW_8B0E.revInfo.REV_AUTHOR := 'M. Gledhill';
   AI_RAW_8B0E.___________0010_0 := false;
   AI_RAW_8B0E.___________0010_1 := false;
   AI_RAW_8B0E.AI_CODE := 16#8B0E;
   AI_RAW_8B0E.___________0020_0 := false;
   AI_RAW_8B0E.___________0020_1 := false;
   AI_RAW_8B0E.RAW_MIN := -5000;
   AI_RAW_8B0E.RAW_MAX := 15000;
   AI_RAW_8B0E.RAW_DESC := 'Thermal Resistance - 3-wire (Cu10 climate - 426)';
   AI_RAW_8B0E.___________0030_1 := false;
   AI_RAW_8B0E.___________0030_2 := false;
   AI_RAW_8B0E.PARAM_TYPE := 16#08;
   AI_RAW_8B0E.PARAM_RANGE := 16#0E;
   AI_RAW_8B0E.PARAM_COEF := 16#0B;
   AI_RAW_8B0E.___________0040_1 := false;
   AI_RAW_8B0E.___________0040_2 := false;
   AI_RAW_8B0E.VALUE_COEF := 0.00426;
   AI_RAW_8C0E.revInfo.REV_BLOCK := 'UT00801';
   AI_RAW_8C0E.revInfo.REV_NUMBER := '001.000';
   AI_RAW_8C0E.revInfo.REV_DATE := '2024-04-09';
   AI_RAW_8C0E.revInfo.REV_AUTHOR := 'M. Gledhill';
   AI_RAW_8C0E.___________0010_0 := false;
   AI_RAW_8C0E.___________0010_1 := false;
   AI_RAW_8C0E.AI_CODE := 16#8C0E;
   AI_RAW_8C0E.___________0020_0 := false;
   AI_RAW_8C0E.___________0020_1 := false;
   AI_RAW_8C0E.RAW_MIN := -5000;
   AI_RAW_8C0E.RAW_MAX := 15000;
   AI_RAW_8C0E.RAW_DESC := 'Thermal Resistance - 3-wire (Cu10 climate - 427)';
   AI_RAW_8C0E.___________0030_1 := false;
   AI_RAW_8C0E.___________0030_2 := false;
   AI_RAW_8C0E.PARAM_TYPE := 16#08;
   AI_RAW_8C0E.PARAM_RANGE := 16#0E;
   AI_RAW_8C0E.PARAM_COEF := 16#0C;
   AI_RAW_8C0E.___________0040_1 := false;
   AI_RAW_8C0E.___________0040_2 := false;
   AI_RAW_8C0E.VALUE_COEF := 0.00427;
   AI_RAW_8D0E.revInfo.REV_BLOCK := 'UT00801';
   AI_RAW_8D0E.revInfo.REV_NUMBER := '001.000';
   AI_RAW_8D0E.revInfo.REV_DATE := '2024-04-09';
   AI_RAW_8D0E.revInfo.REV_AUTHOR := 'M. Gledhill';
   AI_RAW_8D0E.___________0010_0 := false;
   AI_RAW_8D0E.___________0010_1 := false;
   AI_RAW_8D0E.AI_CODE := 16#8D0E;
   AI_RAW_8D0E.___________0020_0 := false;
   AI_RAW_8D0E.___________0020_1 := false;
   AI_RAW_8D0E.RAW_MIN := -5000;
   AI_RAW_8D0E.RAW_MAX := 15000;
   AI_RAW_8D0E.RAW_DESC := 'Thermal Resistance - 3-wire (Cu10 climate - 428)';
   AI_RAW_8D0E.___________0030_1 := false;
   AI_RAW_8D0E.___________0030_2 := false;
   AI_RAW_8D0E.PARAM_TYPE := 16#08;
   AI_RAW_8D0E.PARAM_RANGE := 16#0E;
   AI_RAW_8D0E.PARAM_COEF := 16#0D;
   AI_RAW_8D0E.___________0040_1 := false;
   AI_RAW_8D0E.___________0040_2 := false;
   AI_RAW_8D0E.VALUE_COEF := 0.00428;
   AI_RAW_8B0F.revInfo.REV_BLOCK := 'UT00801';
   AI_RAW_8B0F.revInfo.REV_NUMBER := '001.000';
   AI_RAW_8B0F.revInfo.REV_DATE := '2024-04-09';
   AI_RAW_8B0F.revInfo.REV_AUTHOR := 'M. Gledhill';
   AI_RAW_8B0F.___________0010_0 := false;
   AI_RAW_8B0F.___________0010_1 := false;
   AI_RAW_8B0F.AI_CODE := 16#8B0F;
   AI_RAW_8B0F.___________0020_0 := false;
   AI_RAW_8B0F.___________0020_1 := false;
   AI_RAW_8B0F.RAW_MIN := -500;
   AI_RAW_8B0F.RAW_MAX := 2000;
   AI_RAW_8B0F.RAW_DESC := 'Thermal Resistance - 3-wire (Cu10 standard - 426)';
   AI_RAW_8B0F.___________0030_1 := false;
   AI_RAW_8B0F.___________0030_2 := false;
   AI_RAW_8B0F.PARAM_TYPE := 16#08;
   AI_RAW_8B0F.PARAM_RANGE := 16#0F;
   AI_RAW_8B0F.PARAM_COEF := 16#0B;
   AI_RAW_8B0F.___________0040_1 := false;
   AI_RAW_8B0F.___________0040_2 := false;
   AI_RAW_8B0F.VALUE_COEF := 0.00426;
   AI_RAW_8C0F.revInfo.REV_BLOCK := 'UT00801';
   AI_RAW_8C0F.revInfo.REV_NUMBER := '001.000';
   AI_RAW_8C0F.revInfo.REV_DATE := '2024-04-09';
   AI_RAW_8C0F.revInfo.REV_AUTHOR := 'M. Gledhill';
   AI_RAW_8C0F.___________0010_0 := false;
   AI_RAW_8C0F.___________0010_1 := false;
   AI_RAW_8C0F.AI_CODE := 16#8C0F;
   AI_RAW_8C0F.___________0020_0 := false;
   AI_RAW_8C0F.___________0020_1 := false;
   AI_RAW_8C0F.RAW_MIN := -2000;
   AI_RAW_8C0F.RAW_MAX := 2600;
   AI_RAW_8C0F.RAW_DESC := 'Thermal Resistance - 3-wire (Cu10 standard - 427)';
   AI_RAW_8C0F.___________0030_1 := false;
   AI_RAW_8C0F.___________0030_2 := false;
   AI_RAW_8C0F.PARAM_TYPE := 16#08;
   AI_RAW_8C0F.PARAM_RANGE := 16#0F;
   AI_RAW_8C0F.PARAM_COEF := 16#0C;
   AI_RAW_8C0F.___________0040_1 := false;
   AI_RAW_8C0F.___________0040_2 := false;
   AI_RAW_8C0F.VALUE_COEF := 0.00427;
   AI_RAW_8D0F.revInfo.REV_BLOCK := 'UT00801';
   AI_RAW_8D0F.revInfo.REV_NUMBER := '001.000';
   AI_RAW_8D0F.revInfo.REV_DATE := '2024-04-09';
   AI_RAW_8D0F.revInfo.REV_AUTHOR := 'M. Gledhill';
   AI_RAW_8D0F.___________0010_0 := false;
   AI_RAW_8D0F.___________0010_1 := false;
   AI_RAW_8D0F.AI_CODE := 16#8D0F;
   AI_RAW_8D0F.___________0020_0 := false;
   AI_RAW_8D0F.___________0020_1 := false;
   AI_RAW_8D0F.RAW_MIN := -1800;
   AI_RAW_8D0F.RAW_MAX := 2000;
   AI_RAW_8D0F.RAW_DESC := 'Thermal Resistance - 3-wire (Cu10 standard - 428)';
   AI_RAW_8D0F.___________0030_1 := false;
   AI_RAW_8D0F.___________0030_2 := false;
   AI_RAW_8D0F.PARAM_TYPE := 16#08;
   AI_RAW_8D0F.PARAM_RANGE := 16#0F;
   AI_RAW_8D0F.PARAM_COEF := 16#0D;
   AI_RAW_8D0F.___________0040_1 := false;
   AI_RAW_8D0F.___________0040_2 := false;
   AI_RAW_8D0F.VALUE_COEF := 0.00428;
   AI_RAW_8B19.revInfo.REV_BLOCK := 'UT00801';
   AI_RAW_8B19.revInfo.REV_NUMBER := '001.000';
   AI_RAW_8B19.revInfo.REV_DATE := '2024-04-09';
   AI_RAW_8B19.revInfo.REV_AUTHOR := 'M. Gledhill';
   AI_RAW_8B19.___________0010_0 := false;
   AI_RAW_8B19.___________0010_1 := false;
   AI_RAW_8B19.AI_CODE := 16#8B19;
   AI_RAW_8B19.___________0020_0 := false;
   AI_RAW_8B19.___________0020_1 := false;
   AI_RAW_8B19.RAW_MIN := -5000;
   AI_RAW_8B19.RAW_MAX := 15000;
   AI_RAW_8B19.RAW_DESC := 'Thermal Resistance - 3-wire (Cu50 climate - 426)';
   AI_RAW_8B19.___________0030_1 := false;
   AI_RAW_8B19.___________0030_2 := false;
   AI_RAW_8B19.PARAM_TYPE := 16#08;
   AI_RAW_8B19.PARAM_RANGE := 16#19;
   AI_RAW_8B19.PARAM_COEF := 16#0B;
   AI_RAW_8B19.___________0040_1 := false;
   AI_RAW_8B19.___________0040_2 := false;
   AI_RAW_8B19.VALUE_COEF := 0.00426;
   AI_RAW_8C19.revInfo.REV_BLOCK := 'UT00801';
   AI_RAW_8C19.revInfo.REV_NUMBER := '001.000';
   AI_RAW_8C19.revInfo.REV_DATE := '2024-04-09';
   AI_RAW_8C19.revInfo.REV_AUTHOR := 'M. Gledhill';
   AI_RAW_8C19.___________0010_0 := false;
   AI_RAW_8C19.___________0010_1 := false;
   AI_RAW_8C19.AI_CODE := 16#8C19;
   AI_RAW_8C19.___________0020_0 := false;
   AI_RAW_8C19.___________0020_1 := false;
   AI_RAW_8C19.RAW_MIN := -5000;
   AI_RAW_8C19.RAW_MAX := 15000;
   AI_RAW_8C19.RAW_DESC := 'Thermal Resistance - 3-wire (Cu50 climate - 427)';
   AI_RAW_8C19.___________0030_1 := false;
   AI_RAW_8C19.___________0030_2 := false;
   AI_RAW_8C19.PARAM_TYPE := 16#08;
   AI_RAW_8C19.PARAM_RANGE := 16#19;
   AI_RAW_8C19.PARAM_COEF := 16#0C;
   AI_RAW_8C19.___________0040_1 := false;
   AI_RAW_8C19.___________0040_2 := false;
   AI_RAW_8C19.VALUE_COEF := 0.00427;
   AI_RAW_8D19.revInfo.REV_BLOCK := 'UT00801';
   AI_RAW_8D19.revInfo.REV_NUMBER := '001.000';
   AI_RAW_8D19.revInfo.REV_DATE := '2024-04-09';
   AI_RAW_8D19.revInfo.REV_AUTHOR := 'M. Gledhill';
   AI_RAW_8D19.___________0010_0 := false;
   AI_RAW_8D19.___________0010_1 := false;
   AI_RAW_8D19.AI_CODE := 16#8D19;
   AI_RAW_8D19.___________0020_0 := false;
   AI_RAW_8D19.___________0020_1 := false;
   AI_RAW_8D19.RAW_MIN := -5000;
   AI_RAW_8D19.RAW_MAX := 15000;
   AI_RAW_8D19.RAW_DESC := 'Thermal Resistance - 3-wire (Cu50 climate - 428)';
   AI_RAW_8D19.___________0030_1 := false;
   AI_RAW_8D19.___________0030_2 := false;
   AI_RAW_8D19.PARAM_TYPE := 16#08;
   AI_RAW_8D19.PARAM_RANGE := 16#19;
   AI_RAW_8D19.PARAM_COEF := 16#0D;
   AI_RAW_8D19.___________0040_1 := false;
   AI_RAW_8D19.___________0040_2 := false;
   AI_RAW_8D19.VALUE_COEF := 0.00428;
   AI_RAW_8B18.revInfo.REV_BLOCK := 'UT00801';
   AI_RAW_8B18.revInfo.REV_NUMBER := '001.000';
   AI_RAW_8B18.revInfo.REV_DATE := '2024-04-09';
   AI_RAW_8B18.revInfo.REV_AUTHOR := 'M. Gledhill';
   AI_RAW_8B18.___________0010_0 := false;
   AI_RAW_8B18.___________0010_1 := false;
   AI_RAW_8B18.AI_CODE := 16#8B18;
   AI_RAW_8B18.___________0020_0 := false;
   AI_RAW_8B18.___________0020_1 := false;
   AI_RAW_8B18.RAW_MIN := -500;
   AI_RAW_8B18.RAW_MAX := 2000;
   AI_RAW_8B18.RAW_DESC := 'Thermal Resistance - 3-wire (Cu50 standard - 426)';
   AI_RAW_8B18.___________0030_1 := false;
   AI_RAW_8B18.___________0030_2 := false;
   AI_RAW_8B18.PARAM_TYPE := 16#08;
   AI_RAW_8B18.PARAM_RANGE := 16#18;
   AI_RAW_8B18.PARAM_COEF := 16#0B;
   AI_RAW_8B18.___________0040_1 := false;
   AI_RAW_8B18.___________0040_2 := false;
   AI_RAW_8B18.VALUE_COEF := 0.00426;
   AI_RAW_8C18.revInfo.REV_BLOCK := 'UT00801';
   AI_RAW_8C18.revInfo.REV_NUMBER := '001.000';
   AI_RAW_8C18.revInfo.REV_DATE := '2024-04-09';
   AI_RAW_8C18.revInfo.REV_AUTHOR := 'M. Gledhill';
   AI_RAW_8C18.___________0010_0 := false;
   AI_RAW_8C18.___________0010_1 := false;
   AI_RAW_8C18.AI_CODE := 16#8C18;
   AI_RAW_8C18.___________0020_0 := false;
   AI_RAW_8C18.___________0020_1 := false;
   AI_RAW_8C18.RAW_MIN := -2000;
   AI_RAW_8C18.RAW_MAX := 2600;
   AI_RAW_8C18.RAW_DESC := 'Thermal Resistance - 3-wire (Cu50 standard - 427)';
   AI_RAW_8C18.___________0030_1 := false;
   AI_RAW_8C18.___________0030_2 := false;
   AI_RAW_8C18.PARAM_TYPE := 16#08;
   AI_RAW_8C18.PARAM_RANGE := 16#18;
   AI_RAW_8C18.PARAM_COEF := 16#0C;
   AI_RAW_8C18.___________0040_1 := false;
   AI_RAW_8C18.___________0040_2 := false;
   AI_RAW_8C18.VALUE_COEF := 0.00427;
   AI_RAW_8D18.revInfo.REV_BLOCK := 'UT00801';
   AI_RAW_8D18.revInfo.REV_NUMBER := '001.000';
   AI_RAW_8D18.revInfo.REV_DATE := '2024-04-09';
   AI_RAW_8D18.revInfo.REV_AUTHOR := 'M. Gledhill';
   AI_RAW_8D18.___________0010_0 := false;
   AI_RAW_8D18.___________0010_1 := false;
   AI_RAW_8D18.AI_CODE := 16#8D18;
   AI_RAW_8D18.___________0020_0 := false;
   AI_RAW_8D18.___________0020_1 := false;
   AI_RAW_8D18.RAW_MIN := -1800;
   AI_RAW_8D18.RAW_MAX := 2000;
   AI_RAW_8D18.RAW_DESC := 'Thermal Resistance - 3-wire (Cu50 standard - 428)';
   AI_RAW_8D18.___________0030_1 := false;
   AI_RAW_8D18.___________0030_2 := false;
   AI_RAW_8D18.PARAM_TYPE := 16#08;
   AI_RAW_8D18.PARAM_RANGE := 16#18;
   AI_RAW_8D18.PARAM_COEF := 16#0D;
   AI_RAW_8D18.___________0040_1 := false;
   AI_RAW_8D18.___________0040_2 := false;
   AI_RAW_8D18.VALUE_COEF := 0.00428;
   AI_RAW_8B1B.revInfo.REV_BLOCK := 'UT00801';
   AI_RAW_8B1B.revInfo.REV_NUMBER := '001.000';
   AI_RAW_8B1B.revInfo.REV_DATE := '2024-04-09';
   AI_RAW_8B1B.revInfo.REV_AUTHOR := 'M. Gledhill';
   AI_RAW_8B1B.___________0010_0 := false;
   AI_RAW_8B1B.___________0010_1 := false;
   AI_RAW_8B1B.AI_CODE := 16#8B1B;
   AI_RAW_8B1B.___________0020_0 := false;
   AI_RAW_8B1B.___________0020_1 := false;
   AI_RAW_8B1B.RAW_MIN := -5000;
   AI_RAW_8B1B.RAW_MAX := 15000;
   AI_RAW_8B1B.RAW_DESC := 'Thermal Resistance - 3-wire (Cu100 climate - 426)';
   AI_RAW_8B1B.___________0030_1 := false;
   AI_RAW_8B1B.___________0030_2 := false;
   AI_RAW_8B1B.PARAM_TYPE := 16#08;
   AI_RAW_8B1B.PARAM_RANGE := 16#1B;
   AI_RAW_8B1B.PARAM_COEF := 16#0B;
   AI_RAW_8B1B.___________0040_1 := false;
   AI_RAW_8B1B.___________0040_2 := false;
   AI_RAW_8B1B.VALUE_COEF := 0.00426;
   AI_RAW_8C1B.revInfo.REV_BLOCK := 'UT00801';
   AI_RAW_8C1B.revInfo.REV_NUMBER := '001.000';
   AI_RAW_8C1B.revInfo.REV_DATE := '2024-04-09';
   AI_RAW_8C1B.revInfo.REV_AUTHOR := 'M. Gledhill';
   AI_RAW_8C1B.___________0010_0 := false;
   AI_RAW_8C1B.___________0010_1 := false;
   AI_RAW_8C1B.AI_CODE := 16#8C1B;
   AI_RAW_8C1B.___________0020_0 := false;
   AI_RAW_8C1B.___________0020_1 := false;
   AI_RAW_8C1B.RAW_MIN := -5000;
   AI_RAW_8C1B.RAW_MAX := 15000;
   AI_RAW_8C1B.RAW_DESC := 'Thermal Resistance - 3-wire (Cu100 climate - 427)';
   AI_RAW_8C1B.___________0030_1 := false;
   AI_RAW_8C1B.___________0030_2 := false;
   AI_RAW_8C1B.PARAM_TYPE := 16#08;
   AI_RAW_8C1B.PARAM_RANGE := 16#1B;
   AI_RAW_8C1B.PARAM_COEF := 16#0C;
   AI_RAW_8C1B.___________0040_1 := false;
   AI_RAW_8C1B.___________0040_2 := false;
   AI_RAW_8C1B.VALUE_COEF := 0.00427;
   AI_RAW_8D1B.revInfo.REV_BLOCK := 'UT00801';
   AI_RAW_8D1B.revInfo.REV_NUMBER := '001.000';
   AI_RAW_8D1B.revInfo.REV_DATE := '2024-04-09';
   AI_RAW_8D1B.revInfo.REV_AUTHOR := 'M. Gledhill';
   AI_RAW_8D1B.___________0010_0 := false;
   AI_RAW_8D1B.___________0010_1 := false;
   AI_RAW_8D1B.AI_CODE := 16#8D1B;
   AI_RAW_8D1B.___________0020_0 := false;
   AI_RAW_8D1B.___________0020_1 := false;
   AI_RAW_8D1B.RAW_MIN := -5000;
   AI_RAW_8D1B.RAW_MAX := 15000;
   AI_RAW_8D1B.RAW_DESC := 'Thermal Resistance - 3-wire (Cu100 climate - 428)';
   AI_RAW_8D1B.___________0030_1 := false;
   AI_RAW_8D1B.___________0030_2 := false;
   AI_RAW_8D1B.PARAM_TYPE := 16#08;
   AI_RAW_8D1B.PARAM_RANGE := 16#1B;
   AI_RAW_8D1B.PARAM_COEF := 16#0D;
   AI_RAW_8D1B.___________0040_1 := false;
   AI_RAW_8D1B.___________0040_2 := false;
   AI_RAW_8D1B.VALUE_COEF := 0.00428;
   AI_RAW_8B1A.revInfo.REV_BLOCK := 'UT00801';
   AI_RAW_8B1A.revInfo.REV_NUMBER := '001.000';
   AI_RAW_8B1A.revInfo.REV_DATE := '2024-04-09';
   AI_RAW_8B1A.revInfo.REV_AUTHOR := 'M. Gledhill';
   AI_RAW_8B1A.___________0010_0 := false;
   AI_RAW_8B1A.___________0010_1 := false;
   AI_RAW_8B1A.AI_CODE := 16#8B1A;
   AI_RAW_8B1A.___________0020_0 := false;
   AI_RAW_8B1A.___________0020_1 := false;
   AI_RAW_8B1A.RAW_MIN := -500;
   AI_RAW_8B1A.RAW_MAX := 2000;
   AI_RAW_8B1A.RAW_DESC := 'Thermal Resistance - 3-wire (Cu100 standard - 426)';
   AI_RAW_8B1A.___________0030_1 := false;
   AI_RAW_8B1A.___________0030_2 := false;
   AI_RAW_8B1A.PARAM_TYPE := 16#08;
   AI_RAW_8B1A.PARAM_RANGE := 16#1A;
   AI_RAW_8B1A.PARAM_COEF := 16#0B;
   AI_RAW_8B1A.___________0040_1 := false;
   AI_RAW_8B1A.___________0040_2 := false;
   AI_RAW_8B1A.VALUE_COEF := 0.00426;
   AI_RAW_8C1A.revInfo.REV_BLOCK := 'UT00801';
   AI_RAW_8C1A.revInfo.REV_NUMBER := '001.000';
   AI_RAW_8C1A.revInfo.REV_DATE := '2024-04-09';
   AI_RAW_8C1A.revInfo.REV_AUTHOR := 'M. Gledhill';
   AI_RAW_8C1A.___________0010_0 := false;
   AI_RAW_8C1A.___________0010_1 := false;
   AI_RAW_8C1A.AI_CODE := 16#8C1A;
   AI_RAW_8C1A.___________0020_0 := false;
   AI_RAW_8C1A.___________0020_1 := false;
   AI_RAW_8C1A.RAW_MIN := -2000;
   AI_RAW_8C1A.RAW_MAX := 2600;
   AI_RAW_8C1A.RAW_DESC := 'Thermal Resistance - 3-wire (Cu100 standard - 427)';
   AI_RAW_8C1A.___________0030_1 := false;
   AI_RAW_8C1A.___________0030_2 := false;
   AI_RAW_8C1A.PARAM_TYPE := 16#08;
   AI_RAW_8C1A.PARAM_RANGE := 16#1A;
   AI_RAW_8C1A.PARAM_COEF := 16#0C;
   AI_RAW_8C1A.___________0040_1 := false;
   AI_RAW_8C1A.___________0040_2 := false;
   AI_RAW_8C1A.VALUE_COEF := 0.00427;
   AI_RAW_8D1A.revInfo.REV_BLOCK := 'UT00801';
   AI_RAW_8D1A.revInfo.REV_NUMBER := '001.000';
   AI_RAW_8D1A.revInfo.REV_DATE := '2024-04-09';
   AI_RAW_8D1A.revInfo.REV_AUTHOR := 'M. Gledhill';
   AI_RAW_8D1A.___________0010_0 := false;
   AI_RAW_8D1A.___________0010_1 := false;
   AI_RAW_8D1A.AI_CODE := 16#8D1A;
   AI_RAW_8D1A.___________0020_0 := false;
   AI_RAW_8D1A.___________0020_1 := false;
   AI_RAW_8D1A.RAW_MIN := -1800;
   AI_RAW_8D1A.RAW_MAX := 2000;
   AI_RAW_8D1A.RAW_DESC := 'Thermal Resistance - 3-wire (Cu100 standard - 428)';
   AI_RAW_8D1A.___________0030_1 := false;
   AI_RAW_8D1A.___________0030_2 := false;
   AI_RAW_8D1A.PARAM_TYPE := 16#08;
   AI_RAW_8D1A.PARAM_RANGE := 16#1A;
   AI_RAW_8D1A.PARAM_COEF := 16#0D;
   AI_RAW_8D1A.___________0040_1 := false;
   AI_RAW_8D1A.___________0040_2 := false;
   AI_RAW_8D1A.VALUE_COEF := 0.00428;
   AI_RAW_8A1D.revInfo.REV_BLOCK := 'UT00801';
   AI_RAW_8A1D.revInfo.REV_NUMBER := '001.000';
   AI_RAW_8A1D.revInfo.REV_DATE := '2024-04-09';
   AI_RAW_8A1D.revInfo.REV_AUTHOR := 'M. Gledhill';
   AI_RAW_8A1D.___________0010_0 := false;
   AI_RAW_8A1D.___________0010_1 := false;
   AI_RAW_8A1D.AI_CODE := 16#8A1D;
   AI_RAW_8A1D.___________0020_0 := false;
   AI_RAW_8A1D.___________0020_1 := false;
   AI_RAW_8A1D.RAW_MIN := -6000;
   AI_RAW_8A1D.RAW_MAX := 13000;
   AI_RAW_8A1D.RAW_DESC := 'Thermal Resistance - 3-wire (LG-Ni1000 climate - 500)';
   AI_RAW_8A1D.___________0030_1 := false;
   AI_RAW_8A1D.___________0030_2 := false;
   AI_RAW_8A1D.PARAM_TYPE := 16#08;
   AI_RAW_8A1D.PARAM_RANGE := 16#1D;
   AI_RAW_8A1D.PARAM_COEF := 16#0A;
   AI_RAW_8A1D.___________0040_1 := false;
   AI_RAW_8A1D.___________0040_2 := false;
   AI_RAW_8A1D.VALUE_COEF := 0.005;
   AI_RAW_8A1C.revInfo.REV_BLOCK := 'UT00801';
   AI_RAW_8A1C.revInfo.REV_NUMBER := '001.000';
   AI_RAW_8A1C.revInfo.REV_DATE := '2024-04-09';
   AI_RAW_8A1C.revInfo.REV_AUTHOR := 'M. Gledhill';
   AI_RAW_8A1C.___________0010_0 := false;
   AI_RAW_8A1C.___________0010_1 := false;
   AI_RAW_8A1C.AI_CODE := 16#8A1C;
   AI_RAW_8A1C.___________0020_0 := false;
   AI_RAW_8A1C.___________0020_1 := false;
   AI_RAW_8A1C.RAW_MIN := -600;
   AI_RAW_8A1C.RAW_MAX := 2500;
   AI_RAW_8A1C.RAW_DESC := 'Thermal Resistance - 3-wire (LG-Ni1000 standard - 500)';
   AI_RAW_8A1C.___________0030_1 := false;
   AI_RAW_8A1C.___________0030_2 := false;
   AI_RAW_8A1C.PARAM_TYPE := 16#08;
   AI_RAW_8A1C.PARAM_RANGE := 16#1C;
   AI_RAW_8A1C.PARAM_COEF := 16#0A;
   AI_RAW_8A1C.___________0040_1 := false;
   AI_RAW_8A1C.___________0040_2 := false;
   AI_RAW_8A1C.VALUE_COEF := 0.005;
   AI_RAW_871F.revInfo.REV_BLOCK := 'UT00801';
   AI_RAW_871F.revInfo.REV_NUMBER := '001.000';
   AI_RAW_871F.revInfo.REV_DATE := '2024-04-09';
   AI_RAW_871F.revInfo.REV_AUTHOR := 'M. Gledhill';
   AI_RAW_871F.___________0010_0 := false;
   AI_RAW_871F.___________0010_1 := false;
   AI_RAW_871F.AI_CODE := 16#871F;
   AI_RAW_871F.___________0020_0 := false;
   AI_RAW_871F.___________0020_1 := false;
   AI_RAW_871F.RAW_MIN := -6000;
   AI_RAW_871F.RAW_MAX := 13000;
   AI_RAW_871F.RAW_DESC := 'Thermal Resistance - 3-wire (Ni10 climate - 617)';
   AI_RAW_871F.___________0030_1 := false;
   AI_RAW_871F.___________0030_2 := false;
   AI_RAW_871F.PARAM_TYPE := 16#08;
   AI_RAW_871F.PARAM_RANGE := 16#1F;
   AI_RAW_871F.PARAM_COEF := 16#07;
   AI_RAW_871F.___________0040_1 := false;
   AI_RAW_871F.___________0040_2 := false;
   AI_RAW_871F.VALUE_COEF := 0.00617;
   AI_RAW_881F.revInfo.REV_BLOCK := 'UT00801';
   AI_RAW_881F.revInfo.REV_NUMBER := '001.000';
   AI_RAW_881F.revInfo.REV_DATE := '2024-04-09';
   AI_RAW_881F.revInfo.REV_AUTHOR := 'M. Gledhill';
   AI_RAW_881F.___________0010_0 := false;
   AI_RAW_881F.___________0010_1 := false;
   AI_RAW_881F.AI_CODE := 16#881F;
   AI_RAW_881F.___________0020_0 := false;
   AI_RAW_881F.___________0020_1 := false;
   AI_RAW_881F.RAW_MIN := -6000;
   AI_RAW_881F.RAW_MAX := 13000;
   AI_RAW_881F.RAW_DESC := 'Thermal Resistance - 3-wire (Ni10 climate - 618)';
   AI_RAW_881F.___________0030_1 := false;
   AI_RAW_881F.___________0030_2 := false;
   AI_RAW_881F.PARAM_TYPE := 16#08;
   AI_RAW_881F.PARAM_RANGE := 16#1F;
   AI_RAW_881F.PARAM_COEF := 16#08;
   AI_RAW_881F.___________0040_1 := false;
   AI_RAW_881F.___________0040_2 := false;
   AI_RAW_881F.VALUE_COEF := 0.00618;
   AI_RAW_891F.revInfo.REV_BLOCK := 'UT00801';
   AI_RAW_891F.revInfo.REV_NUMBER := '001.000';
   AI_RAW_891F.revInfo.REV_DATE := '2024-04-09';
   AI_RAW_891F.revInfo.REV_AUTHOR := 'M. Gledhill';
   AI_RAW_891F.___________0010_0 := false;
   AI_RAW_891F.___________0010_1 := false;
   AI_RAW_891F.AI_CODE := 16#891F;
   AI_RAW_891F.___________0020_0 := false;
   AI_RAW_891F.___________0020_1 := false;
   AI_RAW_891F.RAW_MIN := -6000;
   AI_RAW_891F.RAW_MAX := 13000;
   AI_RAW_891F.RAW_DESC := 'Thermal Resistance - 3-wire (Ni10 climate - 672)';
   AI_RAW_891F.___________0030_1 := false;
   AI_RAW_891F.___________0030_2 := false;
   AI_RAW_891F.PARAM_TYPE := 16#08;
   AI_RAW_891F.PARAM_RANGE := 16#1F;
   AI_RAW_891F.PARAM_COEF := 16#09;
   AI_RAW_891F.___________0040_1 := false;
   AI_RAW_891F.___________0040_2 := false;
   AI_RAW_891F.VALUE_COEF := 0.00672;
   AI_RAW_871E.revInfo.REV_BLOCK := 'UT00801';
   AI_RAW_871E.revInfo.REV_NUMBER := '001.000';
   AI_RAW_871E.revInfo.REV_DATE := '2024-04-09';
   AI_RAW_871E.revInfo.REV_AUTHOR := 'M. Gledhill';
   AI_RAW_871E.___________0010_0 := false;
   AI_RAW_871E.___________0010_1 := false;
   AI_RAW_871E.AI_CODE := 16#871E;
   AI_RAW_871E.___________0020_0 := false;
   AI_RAW_871E.___________0020_1 := false;
   AI_RAW_871E.RAW_MIN := -600;
   AI_RAW_871E.RAW_MAX := 1800;
   AI_RAW_871E.RAW_DESC := 'Thermal Resistance - 3-wire (Ni10 standard - 617)';
   AI_RAW_871E.___________0030_1 := false;
   AI_RAW_871E.___________0030_2 := false;
   AI_RAW_871E.PARAM_TYPE := 16#08;
   AI_RAW_871E.PARAM_RANGE := 16#1E;
   AI_RAW_871E.PARAM_COEF := 16#07;
   AI_RAW_871E.___________0040_1 := false;
   AI_RAW_871E.___________0040_2 := false;
   AI_RAW_871E.VALUE_COEF := 0.00617;
   AI_RAW_881E.revInfo.REV_BLOCK := 'UT00801';
   AI_RAW_881E.revInfo.REV_NUMBER := '001.000';
   AI_RAW_881E.revInfo.REV_DATE := '2024-04-09';
   AI_RAW_881E.revInfo.REV_AUTHOR := 'M. Gledhill';
   AI_RAW_881E.___________0010_0 := false;
   AI_RAW_881E.___________0010_1 := false;
   AI_RAW_881E.AI_CODE := 16#881E;
   AI_RAW_881E.___________0020_0 := false;
   AI_RAW_881E.___________0020_1 := false;
   AI_RAW_881E.RAW_MIN := -600;
   AI_RAW_881E.RAW_MAX := 2500;
   AI_RAW_881E.RAW_DESC := 'Thermal Resistance - 3-wire (Ni10 standard - 618)';
   AI_RAW_881E.___________0030_1 := false;
   AI_RAW_881E.___________0030_2 := false;
   AI_RAW_881E.PARAM_TYPE := 16#08;
   AI_RAW_881E.PARAM_RANGE := 16#1E;
   AI_RAW_881E.PARAM_COEF := 16#08;
   AI_RAW_881E.___________0040_1 := false;
   AI_RAW_881E.___________0040_2 := false;
   AI_RAW_881E.VALUE_COEF := 0.00618;
   AI_RAW_891E.revInfo.REV_BLOCK := 'UT00801';
   AI_RAW_891E.revInfo.REV_NUMBER := '001.000';
   AI_RAW_891E.revInfo.REV_DATE := '2024-04-09';
   AI_RAW_891E.revInfo.REV_AUTHOR := 'M. Gledhill';
   AI_RAW_891E.___________0010_0 := false;
   AI_RAW_891E.___________0010_1 := false;
   AI_RAW_891E.AI_CODE := 16#891E;
   AI_RAW_891E.___________0020_0 := false;
   AI_RAW_891E.___________0020_1 := false;
   AI_RAW_891E.RAW_MIN := -600;
   AI_RAW_891E.RAW_MAX := 2500;
   AI_RAW_891E.RAW_DESC := 'Thermal Resistance - 3-wire (Ni10 standard - 672)';
   AI_RAW_891E.___________0030_1 := false;
   AI_RAW_891E.___________0030_2 := false;
   AI_RAW_891E.PARAM_TYPE := 16#08;
   AI_RAW_891E.PARAM_RANGE := 16#1E;
   AI_RAW_891E.PARAM_COEF := 16#09;
   AI_RAW_891E.___________0040_1 := false;
   AI_RAW_891E.___________0040_2 := false;
   AI_RAW_891E.VALUE_COEF := 0.00672;
   AI_RAW_870D.revInfo.REV_BLOCK := 'UT00801';
   AI_RAW_870D.revInfo.REV_NUMBER := '001.000';
   AI_RAW_870D.revInfo.REV_DATE := '2024-04-09';
   AI_RAW_870D.revInfo.REV_AUTHOR := 'M. Gledhill';
   AI_RAW_870D.___________0010_0 := false;
   AI_RAW_870D.___________0010_1 := false;
   AI_RAW_870D.AI_CODE := 16#870D;
   AI_RAW_870D.___________0020_0 := false;
   AI_RAW_870D.___________0020_1 := false;
   AI_RAW_870D.RAW_MIN := -6000;
   AI_RAW_870D.RAW_MAX := 13000;
   AI_RAW_870D.RAW_DESC := 'Thermal Resistance - 3-wire (Ni120 climate - 617)';
   AI_RAW_870D.___________0030_1 := false;
   AI_RAW_870D.___________0030_2 := false;
   AI_RAW_870D.PARAM_TYPE := 16#08;
   AI_RAW_870D.PARAM_RANGE := 16#0D;
   AI_RAW_870D.PARAM_COEF := 16#07;
   AI_RAW_870D.___________0040_1 := false;
   AI_RAW_870D.___________0040_2 := false;
   AI_RAW_870D.VALUE_COEF := 0.00617;
   AI_RAW_880D.revInfo.REV_BLOCK := 'UT00801';
   AI_RAW_880D.revInfo.REV_NUMBER := '001.000';
   AI_RAW_880D.revInfo.REV_DATE := '2024-04-09';
   AI_RAW_880D.revInfo.REV_AUTHOR := 'M. Gledhill';
   AI_RAW_880D.___________0010_0 := false;
   AI_RAW_880D.___________0010_1 := false;
   AI_RAW_880D.AI_CODE := 16#880D;
   AI_RAW_880D.___________0020_0 := false;
   AI_RAW_880D.___________0020_1 := false;
   AI_RAW_880D.RAW_MIN := -6000;
   AI_RAW_880D.RAW_MAX := 13000;
   AI_RAW_880D.RAW_DESC := 'Thermal Resistance - 3-wire (Ni120 climate - 618)';
   AI_RAW_880D.___________0030_1 := false;
   AI_RAW_880D.___________0030_2 := false;
   AI_RAW_880D.PARAM_TYPE := 16#08;
   AI_RAW_880D.PARAM_RANGE := 16#0D;
   AI_RAW_880D.PARAM_COEF := 16#08;
   AI_RAW_880D.___________0040_1 := false;
   AI_RAW_880D.___________0040_2 := false;
   AI_RAW_880D.VALUE_COEF := 0.00618;
   AI_RAW_890D.revInfo.REV_BLOCK := 'UT00801';
   AI_RAW_890D.revInfo.REV_NUMBER := '001.000';
   AI_RAW_890D.revInfo.REV_DATE := '2024-04-09';
   AI_RAW_890D.revInfo.REV_AUTHOR := 'M. Gledhill';
   AI_RAW_890D.___________0010_0 := false;
   AI_RAW_890D.___________0010_1 := false;
   AI_RAW_890D.AI_CODE := 16#890D;
   AI_RAW_890D.___________0020_0 := false;
   AI_RAW_890D.___________0020_1 := false;
   AI_RAW_890D.RAW_MIN := -6000;
   AI_RAW_890D.RAW_MAX := 13000;
   AI_RAW_890D.RAW_DESC := 'Thermal Resistance - 3-wire (Ni120 climate - 672)';
   AI_RAW_890D.___________0030_1 := false;
   AI_RAW_890D.___________0030_2 := false;
   AI_RAW_890D.PARAM_TYPE := 16#08;
   AI_RAW_890D.PARAM_RANGE := 16#0D;
   AI_RAW_890D.PARAM_COEF := 16#09;
   AI_RAW_890D.___________0040_1 := false;
   AI_RAW_890D.___________0040_2 := false;
   AI_RAW_890D.VALUE_COEF := 0.00672;
   AI_RAW_870C.revInfo.REV_BLOCK := 'UT00801';
   AI_RAW_870C.revInfo.REV_NUMBER := '001.000';
   AI_RAW_870C.revInfo.REV_DATE := '2024-04-09';
   AI_RAW_870C.revInfo.REV_AUTHOR := 'M. Gledhill';
   AI_RAW_870C.___________0010_0 := false;
   AI_RAW_870C.___________0010_1 := false;
   AI_RAW_870C.AI_CODE := 16#870C;
   AI_RAW_870C.___________0020_0 := false;
   AI_RAW_870C.___________0020_1 := false;
   AI_RAW_870C.RAW_MIN := -600;
   AI_RAW_870C.RAW_MAX := 1800;
   AI_RAW_870C.RAW_DESC := 'Thermal Resistance - 3-wire (Ni120 standard - 617)';
   AI_RAW_870C.___________0030_1 := false;
   AI_RAW_870C.___________0030_2 := false;
   AI_RAW_870C.PARAM_TYPE := 16#08;
   AI_RAW_870C.PARAM_RANGE := 16#0C;
   AI_RAW_870C.PARAM_COEF := 16#07;
   AI_RAW_870C.___________0040_1 := false;
   AI_RAW_870C.___________0040_2 := false;
   AI_RAW_870C.VALUE_COEF := 0.00617;
   AI_RAW_880C.revInfo.REV_BLOCK := 'UT00801';
   AI_RAW_880C.revInfo.REV_NUMBER := '001.000';
   AI_RAW_880C.revInfo.REV_DATE := '2024-04-09';
   AI_RAW_880C.revInfo.REV_AUTHOR := 'M. Gledhill';
   AI_RAW_880C.___________0010_0 := false;
   AI_RAW_880C.___________0010_1 := false;
   AI_RAW_880C.AI_CODE := 16#880C;
   AI_RAW_880C.___________0020_0 := false;
   AI_RAW_880C.___________0020_1 := false;
   AI_RAW_880C.RAW_MIN := -600;
   AI_RAW_880C.RAW_MAX := 2500;
   AI_RAW_880C.RAW_DESC := 'Thermal Resistance - 3-wire (Ni120 standard - 618)';
   AI_RAW_880C.___________0030_1 := false;
   AI_RAW_880C.___________0030_2 := false;
   AI_RAW_880C.PARAM_TYPE := 16#08;
   AI_RAW_880C.PARAM_RANGE := 16#0C;
   AI_RAW_880C.PARAM_COEF := 16#08;
   AI_RAW_880C.___________0040_1 := false;
   AI_RAW_880C.___________0040_2 := false;
   AI_RAW_880C.VALUE_COEF := 0.00618;
   AI_RAW_890C.revInfo.REV_BLOCK := 'UT00801';
   AI_RAW_890C.revInfo.REV_NUMBER := '001.000';
   AI_RAW_890C.revInfo.REV_DATE := '2024-04-09';
   AI_RAW_890C.revInfo.REV_AUTHOR := 'M. Gledhill';
   AI_RAW_890C.___________0010_0 := false;
   AI_RAW_890C.___________0010_1 := false;
   AI_RAW_890C.AI_CODE := 16#890C;
   AI_RAW_890C.___________0020_0 := false;
   AI_RAW_890C.___________0020_1 := false;
   AI_RAW_890C.RAW_MIN := -600;
   AI_RAW_890C.RAW_MAX := 2500;
   AI_RAW_890C.RAW_DESC := 'Thermal Resistance - 3-wire (Ni120 standard - 672)';
   AI_RAW_890C.___________0030_1 := false;
   AI_RAW_890C.___________0030_2 := false;
   AI_RAW_890C.PARAM_TYPE := 16#08;
   AI_RAW_890C.PARAM_RANGE := 16#0C;
   AI_RAW_890C.PARAM_COEF := 16#09;
   AI_RAW_890C.___________0040_1 := false;
   AI_RAW_890C.___________0040_2 := false;
   AI_RAW_890C.VALUE_COEF := 0.00672;
   AI_RAW_8701.revInfo.REV_BLOCK := 'UT00801';
   AI_RAW_8701.revInfo.REV_NUMBER := '001.000';
   AI_RAW_8701.revInfo.REV_DATE := '2024-04-09';
   AI_RAW_8701.revInfo.REV_AUTHOR := 'M. Gledhill';
   AI_RAW_8701.___________0010_0 := false;
   AI_RAW_8701.___________0010_1 := false;
   AI_RAW_8701.AI_CODE := 16#8701;
   AI_RAW_8701.___________0020_0 := false;
   AI_RAW_8701.___________0020_1 := false;
   AI_RAW_8701.RAW_MIN := -6000;
   AI_RAW_8701.RAW_MAX := 13000;
